REGION Network 4: Alarm_GlobalError SubStation and RemoteIO
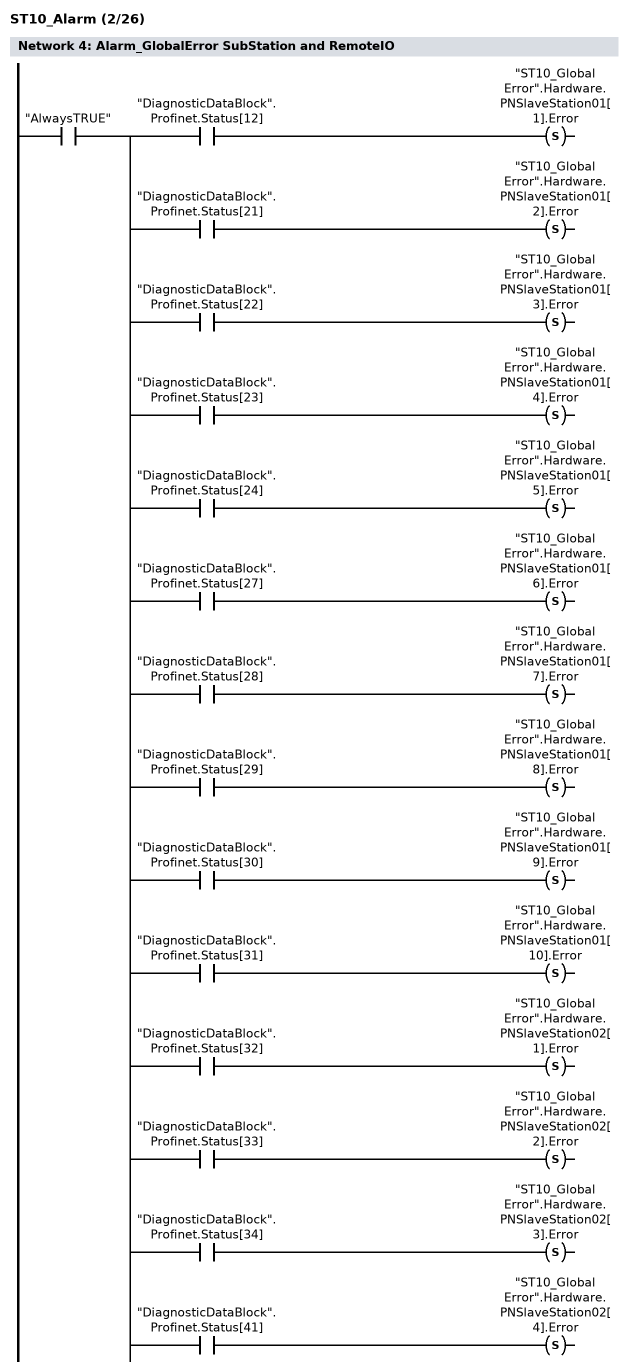
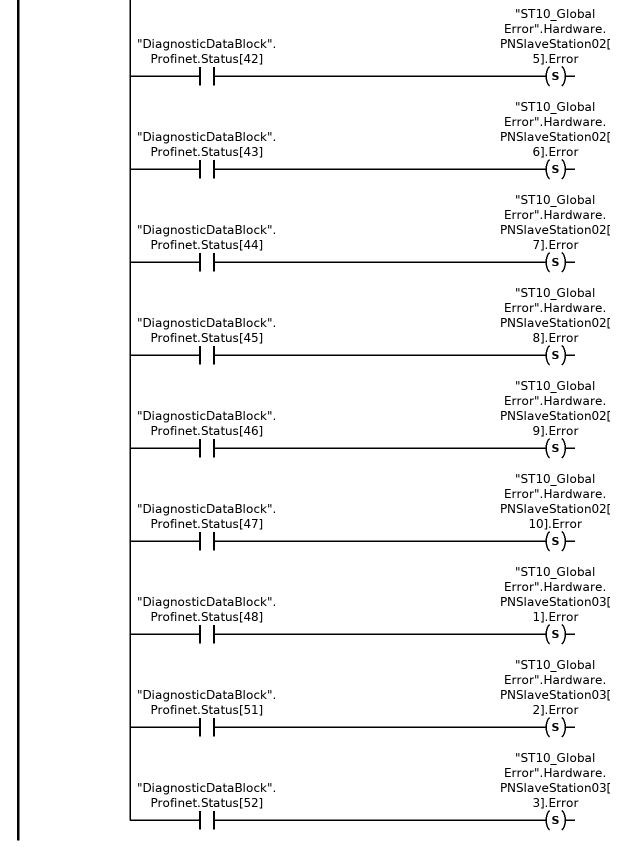
   RUNG wire#powerrail
      Contact( "AlwaysTRUE" )
      wire#w1
      Contact( "DiagnosticDataBlock".Profinet.Status[12] )
      S_Coil( "ST10_GlobalError".Hardware.PNSlaveStation01[1].Error )
   END_RUNG
   RUNG wire#w1
      Contact( "DiagnosticDataBlock".Profinet.Status[21] )
      S_Coil( "ST10_GlobalError".Hardware.PNSlaveStation01[2].Error )
   END_RUNG
   RUNG wire#w1
      Contact( "DiagnosticDataBlock".Profinet.Status[22] )
      S_Coil( "ST10_GlobalError".Hardware.PNSlaveStation01[3].Error )
   END_RUNG
   RUNG wire#w1
      Contact( "DiagnosticDataBlock".Profinet.Status[23] )
      S_Coil( "ST10_GlobalError".Hardware.PNSlaveStation01[4].Error )
   END_RUNG
   RUNG wire#w1
      Contact( "DiagnosticDataBlock".Profinet.Status[24] )
      S_Coil( "ST10_GlobalError".Hardware.PNSlaveStation01[5].Error )
   END_RUNG
   RUNG wire#w1
      Contact( "DiagnosticDataBlock".Profinet.Status[27] )
      S_Coil( "ST10_GlobalError".Hardware.PNSlaveStation01[6].Error )
   END_RUNG
   RUNG wire#w1
      Contact( "DiagnosticDataBlock".Profinet.Status[28] )
      S_Coil( "ST10_GlobalError".Hardware.PNSlaveStation01[7].Error )
   END_RUNG
   RUNG wire#w1
      Contact( "DiagnosticDataBlock".Profinet.Status[29] )
      S_Coil( "ST10_GlobalError".Hardware.PNSlaveStation01[8].Error )
   END_RUNG
   RUNG wire#w1
      Contact( "DiagnosticDataBlock".Profinet.Status[30] )
      S_Coil( "ST10_GlobalError".Hardware.PNSlaveStation01[9].Error )
   END_RUNG
   RUNG wire#w1
      Contact( "DiagnosticDataBlock".Profinet.Status[31] )
      S_Coil( "ST10_GlobalError".Hardware.PNSlaveStation01[10].Error )
   END_RUNG
   RUNG wire#w1
      Contact( "DiagnosticDataBlock".Profinet.Status[32] )
      S_Coil( "ST10_GlobalError".Hardware.PNSlaveStation02[1].Error )
   END_RUNG
   RUNG wire#w1
      Contact( "DiagnosticDataBlock".Profinet.Status[33] )
      S_Coil( "ST10_GlobalError".Hardware.PNSlaveStation02[2].Error )
   END_RUNG
   RUNG wire#w1
      Contact( "DiagnosticDataBlock".Profinet.Status[34] )
      S_Coil( "ST10_GlobalError".Hardware.PNSlaveStation02[3].Error )
   END_RUNG
   RUNG wire#w1
      Contact( "DiagnosticDataBlock".Profinet.Status[41] )
      S_Coil( "ST10_GlobalError".Hardware.PNSlaveStation02[4].Error )
   END_RUNG
   RUNG wire#w1
      Contact( "DiagnosticDataBlock".Profinet.Status[42] )
      S_Coil( "ST10_GlobalError".Hardware.PNSlaveStation02[5].Error )
   END_RUNG
   RUNG wire#w1
      Contact( "DiagnosticDataBlock".Profinet.Status[43] )
      S_Coil( "ST10_GlobalError".Hardware.PNSlaveStation02[6].Error )
   END_RUNG
   RUNG wire#w1
      Contact( "DiagnosticDataBlock".Profinet.Status[44] )
      S_Coil( "ST10_GlobalError".Hardware.PNSlaveStation02[7].Error )
   END_RUNG
   RUNG wire#w1
      Contact( "DiagnosticDataBlock".Profinet.Status[45] )
      S_Coil( "ST10_GlobalError".Hardware.PNSlaveStation02[8].Error )
   END_RUNG
   RUNG wire#w1
      Contact( "DiagnosticDataBlock".Profinet.Status[46] )
      S_Coil( "ST10_GlobalError".Hardware.PNSlaveStation02[9].Error )
   END_RUNG
   RUNG wire#w1
      Contact( "DiagnosticDataBlock".Profinet.Status[47] )
      S_Coil( "ST10_GlobalError".Hardware.PNSlaveStation02[10].Error )
   END_RUNG
   RUNG wire#w1
      Contact( "DiagnosticDataBlock".Profinet.Status[48] )
      S_Coil( "ST10_GlobalError".Hardware.PNSlaveStation03[1].Error )
   END_RUNG
   RUNG wire#w1
      Contact( "DiagnosticDataBlock".Profinet.Status[51] )
      S_Coil( "ST10_GlobalError".Hardware.PNSlaveStation03[2].Error )
   END_RUNG
   RUNG wire#w1
      Contact( "DiagnosticDataBlock".Profinet.Status[52] )
      S_Coil( "ST10_GlobalError".Hardware.PNSlaveStation03[3].Error )
   END_RUNG
   // the same network as SCL:
   IF "AlwaysTRUE" AND "DiagnosticDataBlock".Profinet.Status[12] THEN
       "ST10_GlobalError".Hardware.PNSlaveStation01[1].Error := TRUE;
   END_IF;
   IF "AlwaysTRUE" AND "DiagnosticDataBlock".Profinet.Status[21] THEN
       "ST10_GlobalError".Hardware.PNSlaveStation01[2].Error := TRUE;
   END_IF;
   IF "AlwaysTRUE" AND "DiagnosticDataBlock".Profinet.Status[22] THEN
       "ST10_GlobalError".Hardware.PNSlaveStation01[3].Error := TRUE;
   END_IF;
   IF "AlwaysTRUE" AND "DiagnosticDataBlock".Profinet.Status[23] THEN
       "ST10_GlobalError".Hardware.PNSlaveStation01[4].Error := TRUE;
   END_IF;
   IF "AlwaysTRUE" AND "DiagnosticDataBlock".Profinet.Status[24] THEN
       "ST10_GlobalError".Hardware.PNSlaveStation01[5].Error := TRUE;
   END_IF;
   IF "AlwaysTRUE" AND "DiagnosticDataBlock".Profinet.Status[27] THEN
       "ST10_GlobalError".Hardware.PNSlaveStation01[6].Error := TRUE;
   END_IF;
   IF "AlwaysTRUE" AND "DiagnosticDataBlock".Profinet.Status[28] THEN
       "ST10_GlobalError".Hardware.PNSlaveStation01[7].Error := TRUE;
   END_IF;
   IF "AlwaysTRUE" AND "DiagnosticDataBlock".Profinet.Status[29] THEN
       "ST10_GlobalError".Hardware.PNSlaveStation01[8].Error := TRUE;
   END_IF;
   IF "AlwaysTRUE" AND "DiagnosticDataBlock".Profinet.Status[30] THEN
       "ST10_GlobalError".Hardware.PNSlaveStation01[9].Error := TRUE;
   END_IF;
   IF "AlwaysTRUE" AND "DiagnosticDataBlock".Profinet.Status[31] THEN
       "ST10_GlobalError".Hardware.PNSlaveStation01[10].Error := TRUE;
   END_IF;
   IF "AlwaysTRUE" AND "DiagnosticDataBlock".Profinet.Status[32] THEN
       "ST10_GlobalError".Hardware.PNSlaveStation02[1].Error := TRUE;
   END_IF;
   IF "AlwaysTRUE" AND "DiagnosticDataBlock".Profinet.Status[33] THEN
       "ST10_GlobalError".Hardware.PNSlaveStation02[2].Error := TRUE;
   END_IF;
   IF "AlwaysTRUE" AND "DiagnosticDataBlock".Profinet.Status[34] THEN
       "ST10_GlobalError".Hardware.PNSlaveStation02[3].Error := TRUE;
   END_IF;
   IF "AlwaysTRUE" AND "DiagnosticDataBlock".Profinet.Status[41] THEN
       "ST10_GlobalError".Hardware.PNSlaveStation02[4].Error := TRUE;
   END_IF;
   IF "AlwaysTRUE" AND "DiagnosticDataBlock".Profinet.Status[42] THEN
       "ST10_GlobalError".Hardware.PNSlaveStation02[5].Error := TRUE;
   END_IF;
   IF "AlwaysTRUE" AND "DiagnosticDataBlock".Profinet.Status[43] THEN
       "ST10_GlobalError".Hardware.PNSlaveStation02[6].Error := TRUE;
   END_IF;
   IF "AlwaysTRUE" AND "DiagnosticDataBlock".Profinet.Status[44] THEN
       "ST10_GlobalError".Hardware.PNSlaveStation02[7].Error := TRUE;
   END_IF;
   IF "AlwaysTRUE" AND "DiagnosticDataBlock".Profinet.Status[45] THEN
       "ST10_GlobalError".Hardware.PNSlaveStation02[8].Error := TRUE;
   END_IF;
   IF "AlwaysTRUE" AND "DiagnosticDataBlock".Profinet.Status[46] THEN
       "ST10_GlobalError".Hardware.PNSlaveStation02[9].Error := TRUE;
   END_IF;
   IF "AlwaysTRUE" AND "DiagnosticDataBlock".Profinet.Status[47] THEN
       "ST10_GlobalError".Hardware.PNSlaveStation02[10].Error := TRUE;
   END_IF;
   IF "AlwaysTRUE" AND "DiagnosticDataBlock".Profinet.Status[48] THEN
       "ST10_GlobalError".Hardware.PNSlaveStation03[1].Error := TRUE;
   END_IF;
   IF "AlwaysTRUE" AND "DiagnosticDataBlock".Profinet.Status[51] THEN
       "ST10_GlobalError".Hardware.PNSlaveStation03[2].Error := TRUE;
   END_IF;
   IF "AlwaysTRUE" AND "DiagnosticDataBlock".Profinet.Status[52] THEN
       "ST10_GlobalError".Hardware.PNSlaveStation03[3].Error := TRUE;
   END_IF;
END_REGION

REGION Network 5: Alarm_GlobalError Valve island
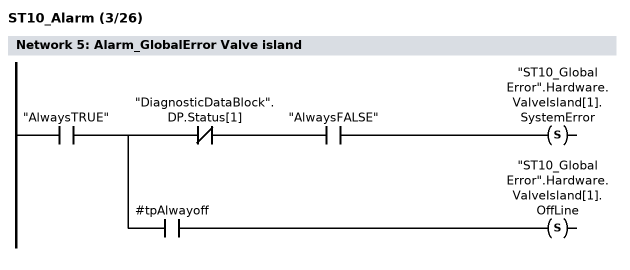
   RUNG wire#powerrail
      Contact( "AlwaysTRUE" )
      wire#w1
      I_Contact( "DiagnosticDataBlock".DP.Status[1] )
      Contact( "AlwaysFALSE" )
      S_Coil( "ST10_GlobalError".Hardware.ValveIsland[1].SystemError )
   END_RUNG
   RUNG wire#w1
      Contact( #tpAlwayoff )
      S_Coil( "ST10_GlobalError".Hardware.ValveIsland[1].OffLine )
   END_RUNG
   // the same network as SCL:
   IF "AlwaysTRUE" AND NOT "DiagnosticDataBlock".DP.Status[1] AND "AlwaysFALSE" THEN
       "ST10_GlobalError".Hardware.ValveIsland[1].SystemError := TRUE;
   END_IF;
   IF "AlwaysTRUE" AND #tpAlwayoff THEN "ST10_GlobalError".Hardware.ValveIsland[1].OffLine := TRUE; END_IF;
END_REGION

REGION Network 6: Alarm_GlobalError Safety Circuit and E-stop
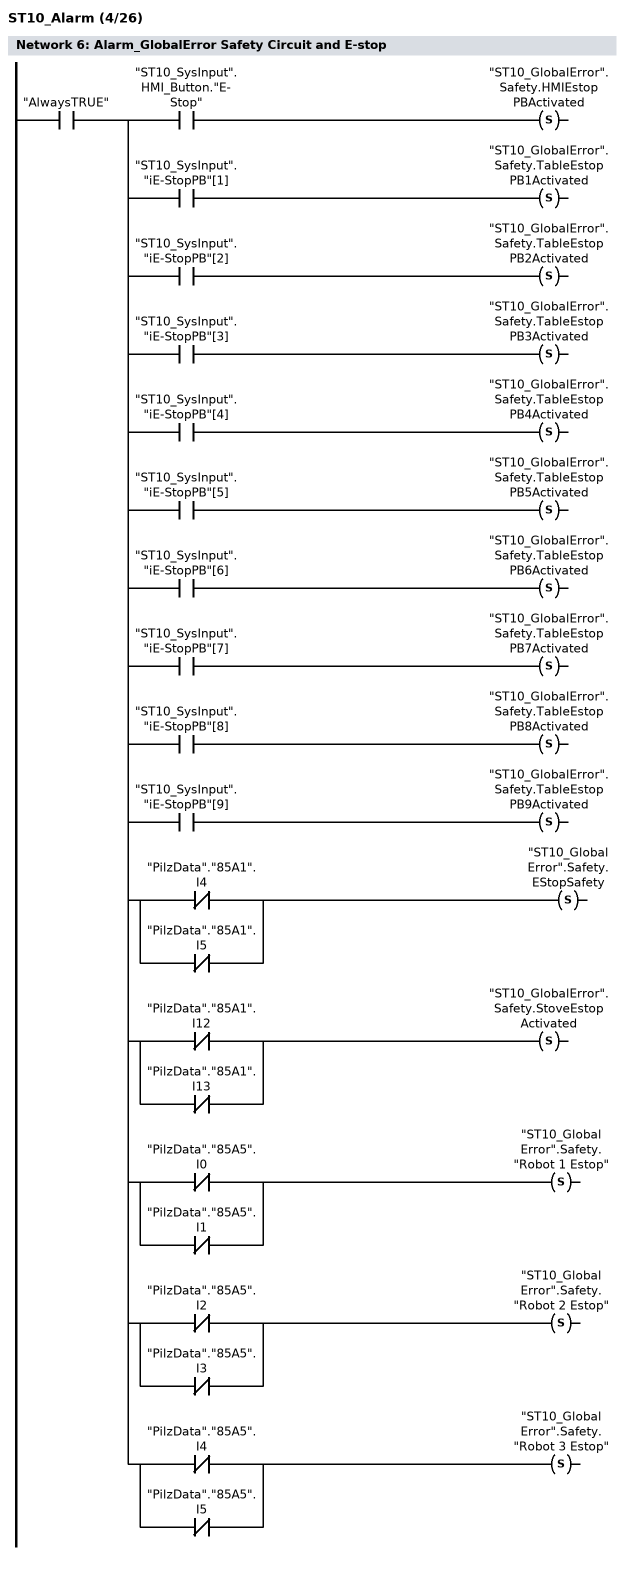
   RUNG wire#powerrail
      Contact( "AlwaysTRUE" )
      wire#w1
      Contact( "ST10_SysInput".HMI_Button."E-Stop" )
      S_Coil( "ST10_GlobalError".Safety.HMIEstopPBActivated )
   END_RUNG
   RUNG wire#w1
      Contact( "ST10_SysInput"."iE-StopPB"[1] )
      S_Coil( "ST10_GlobalError".Safety.TableEstopPB1Activated )
   END_RUNG
   RUNG wire#w1
      Contact( "ST10_SysInput"."iE-StopPB"[2] )
      S_Coil( "ST10_GlobalError".Safety.TableEstopPB2Activated )
   END_RUNG
   RUNG wire#w1
      Contact( "ST10_SysInput"."iE-StopPB"[3] )
      S_Coil( "ST10_GlobalError".Safety.TableEstopPB3Activated )
   END_RUNG
   RUNG wire#w1
      Contact( "ST10_SysInput"."iE-StopPB"[4] )
      S_Coil( "ST10_GlobalError".Safety.TableEstopPB4Activated )
   END_RUNG
   RUNG wire#w1
      Contact( "ST10_SysInput"."iE-StopPB"[5] )
      S_Coil( "ST10_GlobalError".Safety.TableEstopPB5Activated )
   END_RUNG
   RUNG wire#w1
      Contact( "ST10_SysInput"."iE-StopPB"[6] )
      S_Coil( "ST10_GlobalError".Safety.TableEstopPB6Activated )
   END_RUNG
   RUNG wire#w1
      Contact( "ST10_SysInput"."iE-StopPB"[7] )
      S_Coil( "ST10_GlobalError".Safety.TableEstopPB7Activated )
   END_RUNG
   RUNG wire#w1
      Contact( "ST10_SysInput"."iE-StopPB"[8] )
      S_Coil( "ST10_GlobalError".Safety.TableEstopPB8Activated )
   END_RUNG
   RUNG wire#w1
      Contact( "ST10_SysInput"."iE-StopPB"[9] )
      S_Coil( "ST10_GlobalError".Safety.TableEstopPB9Activated )
   END_RUNG
   RUNG wire#w1
      I_Contact( "PilzData"."85A1".I4 )
      wire#w2
      S_Coil( "ST10_GlobalError".Safety.EStopSafety )
   END_RUNG
   RUNG wire#w1
      I_Contact( "PilzData"."85A1".I5 )
   END_RUNG wire#w2
   RUNG wire#w1
      I_Contact( "PilzData"."85A1".I12 )
      wire#w3
      S_Coil( "ST10_GlobalError".Safety.StoveEstopActivated )
   END_RUNG
   RUNG wire#w1
      I_Contact( "PilzData"."85A1".I13 )
   END_RUNG wire#w3
   RUNG wire#w1
      I_Contact( "PilzData"."85A5".I0 )
      wire#w4
      S_Coil( "ST10_GlobalError".Safety."Robot 1 Estop" )
   END_RUNG
   RUNG wire#w1
      I_Contact( "PilzData"."85A5".I1 )
   END_RUNG wire#w4
   RUNG wire#w1
      I_Contact( "PilzData"."85A5".I2 )
      wire#w5
      S_Coil( "ST10_GlobalError".Safety."Robot 2 Estop" )
   END_RUNG
   RUNG wire#w1
      I_Contact( "PilzData"."85A5".I3 )
   END_RUNG wire#w5
   RUNG wire#w1
      I_Contact( "PilzData"."85A5".I4 )
      wire#w6
      S_Coil( "ST10_GlobalError".Safety."Robot 3 Estop" )
   END_RUNG
   RUNG wire#w1
      I_Contact( "PilzData"."85A5".I5 )
   END_RUNG wire#w6
   // the same network as SCL:
   IF "AlwaysTRUE" AND "ST10_SysInput".HMI_Button."E-Stop" THEN
       "ST10_GlobalError".Safety.HMIEstopPBActivated := TRUE;
   END_IF;
   IF "AlwaysTRUE" AND "ST10_SysInput"."iE-StopPB"[1] THEN
       "ST10_GlobalError".Safety.TableEstopPB1Activated := TRUE;
   END_IF;
   IF "AlwaysTRUE" AND "ST10_SysInput"."iE-StopPB"[2] THEN
       "ST10_GlobalError".Safety.TableEstopPB2Activated := TRUE;
   END_IF;
   IF "AlwaysTRUE" AND "ST10_SysInput"."iE-StopPB"[3] THEN
       "ST10_GlobalError".Safety.TableEstopPB3Activated := TRUE;
   END_IF;
   IF "AlwaysTRUE" AND "ST10_SysInput"."iE-StopPB"[4] THEN
       "ST10_GlobalError".Safety.TableEstopPB4Activated := TRUE;
   END_IF;
   IF "AlwaysTRUE" AND "ST10_SysInput"."iE-StopPB"[5] THEN
       "ST10_GlobalError".Safety.TableEstopPB5Activated := TRUE;
   END_IF;
   IF "AlwaysTRUE" AND "ST10_SysInput"."iE-StopPB"[6] THEN
       "ST10_GlobalError".Safety.TableEstopPB6Activated := TRUE;
   END_IF;
   IF "AlwaysTRUE" AND "ST10_SysInput"."iE-StopPB"[7] THEN
       "ST10_GlobalError".Safety.TableEstopPB7Activated := TRUE;
   END_IF;
   IF "AlwaysTRUE" AND "ST10_SysInput"."iE-StopPB"[8] THEN
       "ST10_GlobalError".Safety.TableEstopPB8Activated := TRUE;
   END_IF;
   IF "AlwaysTRUE" AND "ST10_SysInput"."iE-StopPB"[9] THEN
       "ST10_GlobalError".Safety.TableEstopPB9Activated := TRUE;
   END_IF;
   IF "AlwaysTRUE" AND (NOT "PilzData"."85A1".I4 OR NOT "PilzData"."85A1".I5) THEN
       "ST10_GlobalError".Safety.EStopSafety := TRUE;
   END_IF;
   IF "AlwaysTRUE" AND (NOT "PilzData"."85A1".I12 OR NOT "PilzData"."85A1".I13) THEN
       "ST10_GlobalError".Safety.StoveEstopActivated := TRUE;
   END_IF;
   IF "AlwaysTRUE" AND (NOT "PilzData"."85A5".I0 OR NOT "PilzData"."85A5".I1) THEN
       "ST10_GlobalError".Safety."Robot 1 Estop" := TRUE;
   END_IF;
   IF "AlwaysTRUE" AND (NOT "PilzData"."85A5".I2 OR NOT "PilzData"."85A5".I3) THEN
       "ST10_GlobalError".Safety."Robot 2 Estop" := TRUE;
   END_IF;
   IF "AlwaysTRUE" AND (NOT "PilzData"."85A5".I4 OR NOT "PilzData"."85A5".I5) THEN
       "ST10_GlobalError".Safety."Robot 3 Estop" := TRUE;
   END_IF;
END_REGION

REGION Network 7: Alarm_GlobalError Safety Door / Alarm_GlobalError Safety Door 110-124
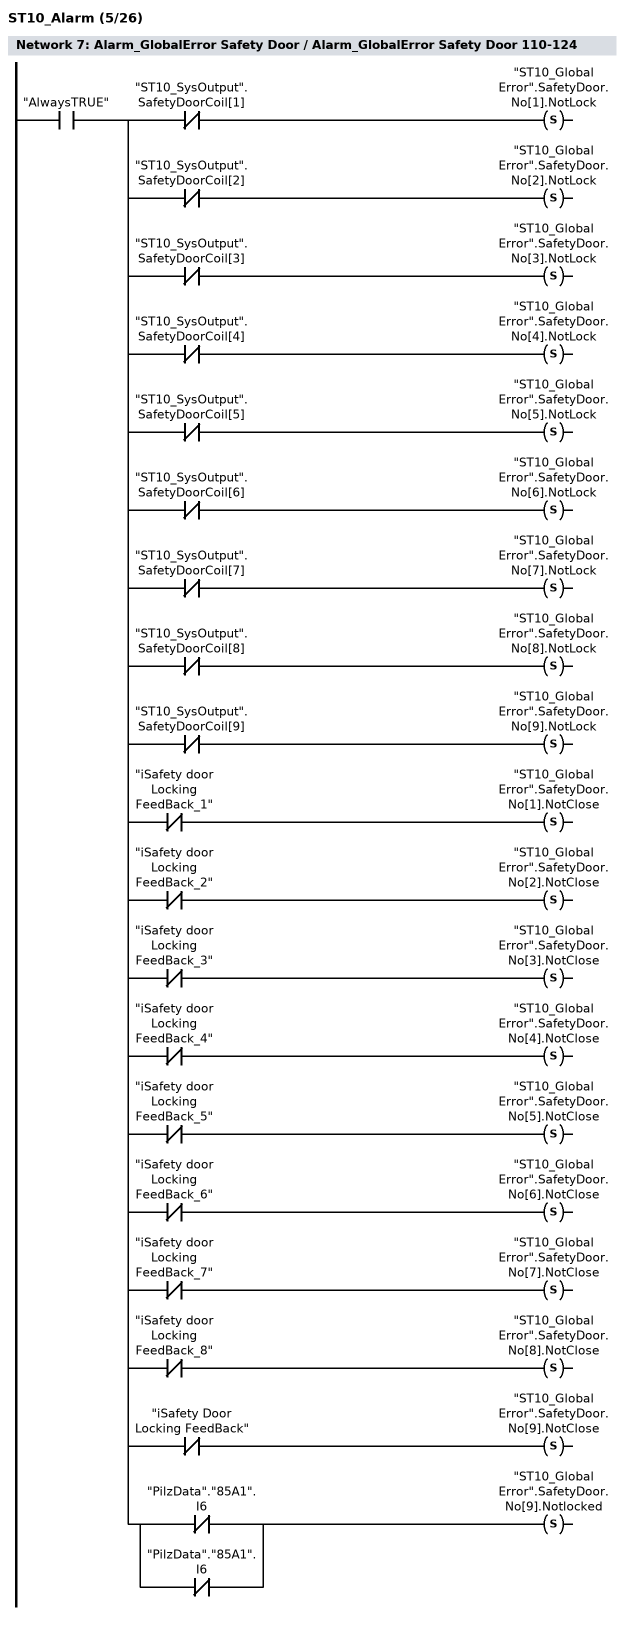
   RUNG wire#powerrail
      Contact( "AlwaysTRUE" )
      wire#w1
      I_Contact( "ST10_SysOutput".SafetyDoorCoil[1] )
      S_Coil( "ST10_GlobalError".SafetyDoor.No[1].NotLock )
   END_RUNG
   RUNG wire#w1
      I_Contact( "ST10_SysOutput".SafetyDoorCoil[2] )
      S_Coil( "ST10_GlobalError".SafetyDoor.No[2].NotLock )
   END_RUNG
   RUNG wire#w1
      I_Contact( "ST10_SysOutput".SafetyDoorCoil[3] )
      S_Coil( "ST10_GlobalError".SafetyDoor.No[3].NotLock )
   END_RUNG
   RUNG wire#w1
      I_Contact( "ST10_SysOutput".SafetyDoorCoil[4] )
      S_Coil( "ST10_GlobalError".SafetyDoor.No[4].NotLock )
   END_RUNG
   RUNG wire#w1
      I_Contact( "ST10_SysOutput".SafetyDoorCoil[5] )
      S_Coil( "ST10_GlobalError".SafetyDoor.No[5].NotLock )
   END_RUNG
   RUNG wire#w1
      I_Contact( "ST10_SysOutput".SafetyDoorCoil[6] )
      S_Coil( "ST10_GlobalError".SafetyDoor.No[6].NotLock )
   END_RUNG
   RUNG wire#w1
      I_Contact( "ST10_SysOutput".SafetyDoorCoil[7] )
      S_Coil( "ST10_GlobalError".SafetyDoor.No[7].NotLock )
   END_RUNG
   RUNG wire#w1
      I_Contact( "ST10_SysOutput".SafetyDoorCoil[8] )
      S_Coil( "ST10_GlobalError".SafetyDoor.No[8].NotLock )
   END_RUNG
   RUNG wire#w1
      I_Contact( "ST10_SysOutput".SafetyDoorCoil[9] )
      S_Coil( "ST10_GlobalError".SafetyDoor.No[9].NotLock )
   END_RUNG
   RUNG wire#w1
      I_Contact( "iSafety door Locking FeedBack_1" )
      S_Coil( "ST10_GlobalError".SafetyDoor.No[1].NotClose )
   END_RUNG
   RUNG wire#w1
      I_Contact( "iSafety door Locking FeedBack_2" )
      S_Coil( "ST10_GlobalError".SafetyDoor.No[2].NotClose )
   END_RUNG
   RUNG wire#w1
      I_Contact( "iSafety door Locking FeedBack_3" )
      S_Coil( "ST10_GlobalError".SafetyDoor.No[3].NotClose )
   END_RUNG
   RUNG wire#w1
      I_Contact( "iSafety door Locking FeedBack_4" )
      S_Coil( "ST10_GlobalError".SafetyDoor.No[4].NotClose )
   END_RUNG
   RUNG wire#w1
      I_Contact( "iSafety door Locking FeedBack_5" )
      S_Coil( "ST10_GlobalError".SafetyDoor.No[5].NotClose )
   END_RUNG
   RUNG wire#w1
      I_Contact( "iSafety door Locking FeedBack_6" )
      S_Coil( "ST10_GlobalError".SafetyDoor.No[6].NotClose )
   END_RUNG
   RUNG wire#w1
      I_Contact( "iSafety door Locking FeedBack_7" )
      S_Coil( "ST10_GlobalError".SafetyDoor.No[7].NotClose )
   END_RUNG
   RUNG wire#w1
      I_Contact( "iSafety door Locking FeedBack_8" )
      S_Coil( "ST10_GlobalError".SafetyDoor.No[8].NotClose )
   END_RUNG
   RUNG wire#w1
      I_Contact( "iSafety Door Locking FeedBack" )
      S_Coil( "ST10_GlobalError".SafetyDoor.No[9].NotClose )
   END_RUNG
   RUNG wire#w1
      I_Contact( "PilzData"."85A1".I6 )
      wire#w2
      S_Coil( "ST10_GlobalError".SafetyDoor.No[9].Notlocked )
   END_RUNG
   RUNG wire#w1
      I_Contact( "PilzData"."85A1".I6 )
   END_RUNG wire#w2
   // the same network as SCL:
   IF "AlwaysTRUE" AND NOT "ST10_SysOutput".SafetyDoorCoil[1] THEN
       "ST10_GlobalError".SafetyDoor.No[1].NotLock := TRUE;
   END_IF;
   IF "AlwaysTRUE" AND NOT "ST10_SysOutput".SafetyDoorCoil[2] THEN
       "ST10_GlobalError".SafetyDoor.No[2].NotLock := TRUE;
   END_IF;
   IF "AlwaysTRUE" AND NOT "ST10_SysOutput".SafetyDoorCoil[3] THEN
       "ST10_GlobalError".SafetyDoor.No[3].NotLock := TRUE;
   END_IF;
   IF "AlwaysTRUE" AND NOT "ST10_SysOutput".SafetyDoorCoil[4] THEN
       "ST10_GlobalError".SafetyDoor.No[4].NotLock := TRUE;
   END_IF;
   IF "AlwaysTRUE" AND NOT "ST10_SysOutput".SafetyDoorCoil[5] THEN
       "ST10_GlobalError".SafetyDoor.No[5].NotLock := TRUE;
   END_IF;
   IF "AlwaysTRUE" AND NOT "ST10_SysOutput".SafetyDoorCoil[6] THEN
       "ST10_GlobalError".SafetyDoor.No[6].NotLock := TRUE;
   END_IF;
   IF "AlwaysTRUE" AND NOT "ST10_SysOutput".SafetyDoorCoil[7] THEN
       "ST10_GlobalError".SafetyDoor.No[7].NotLock := TRUE;
   END_IF;
   IF "AlwaysTRUE" AND NOT "ST10_SysOutput".SafetyDoorCoil[8] THEN
       "ST10_GlobalError".SafetyDoor.No[8].NotLock := TRUE;
   END_IF;
   IF "AlwaysTRUE" AND NOT "ST10_SysOutput".SafetyDoorCoil[9] THEN
       "ST10_GlobalError".SafetyDoor.No[9].NotLock := TRUE;
   END_IF;
   IF "AlwaysTRUE" AND NOT "iSafety door Locking FeedBack_1" THEN
       "ST10_GlobalError".SafetyDoor.No[1].NotClose := TRUE;
   END_IF;
   IF "AlwaysTRUE" AND NOT "iSafety door Locking FeedBack_2" THEN
       "ST10_GlobalError".SafetyDoor.No[2].NotClose := TRUE;
   END_IF;
   IF "AlwaysTRUE" AND NOT "iSafety door Locking FeedBack_3" THEN
       "ST10_GlobalError".SafetyDoor.No[3].NotClose := TRUE;
   END_IF;
   IF "AlwaysTRUE" AND NOT "iSafety door Locking FeedBack_4" THEN
       "ST10_GlobalError".SafetyDoor.No[4].NotClose := TRUE;
   END_IF;
   IF "AlwaysTRUE" AND NOT "iSafety door Locking FeedBack_5" THEN
       "ST10_GlobalError".SafetyDoor.No[5].NotClose := TRUE;
   END_IF;
   IF "AlwaysTRUE" AND NOT "iSafety door Locking FeedBack_6" THEN
       "ST10_GlobalError".SafetyDoor.No[6].NotClose := TRUE;
   END_IF;
   IF "AlwaysTRUE" AND NOT "iSafety door Locking FeedBack_7" THEN
       "ST10_GlobalError".SafetyDoor.No[7].NotClose := TRUE;
   END_IF;
   IF "AlwaysTRUE" AND NOT "iSafety door Locking FeedBack_8" THEN
       "ST10_GlobalError".SafetyDoor.No[8].NotClose := TRUE;
   END_IF;
   IF "AlwaysTRUE" AND NOT "iSafety Door Locking FeedBack" THEN
       "ST10_GlobalError".SafetyDoor.No[9].NotClose := TRUE;
   END_IF;
   IF "AlwaysTRUE" AND (NOT "PilzData"."85A1".I6 OR NOT "PilzData"."85A1".I6) THEN
       "ST10_GlobalError".SafetyDoor.No[9].Notlocked := TRUE;
   END_IF;
END_REGION

REGION Network 8: Alarm_GlobalError Safety Door / Alarm_GlobalError Material Door 128-129
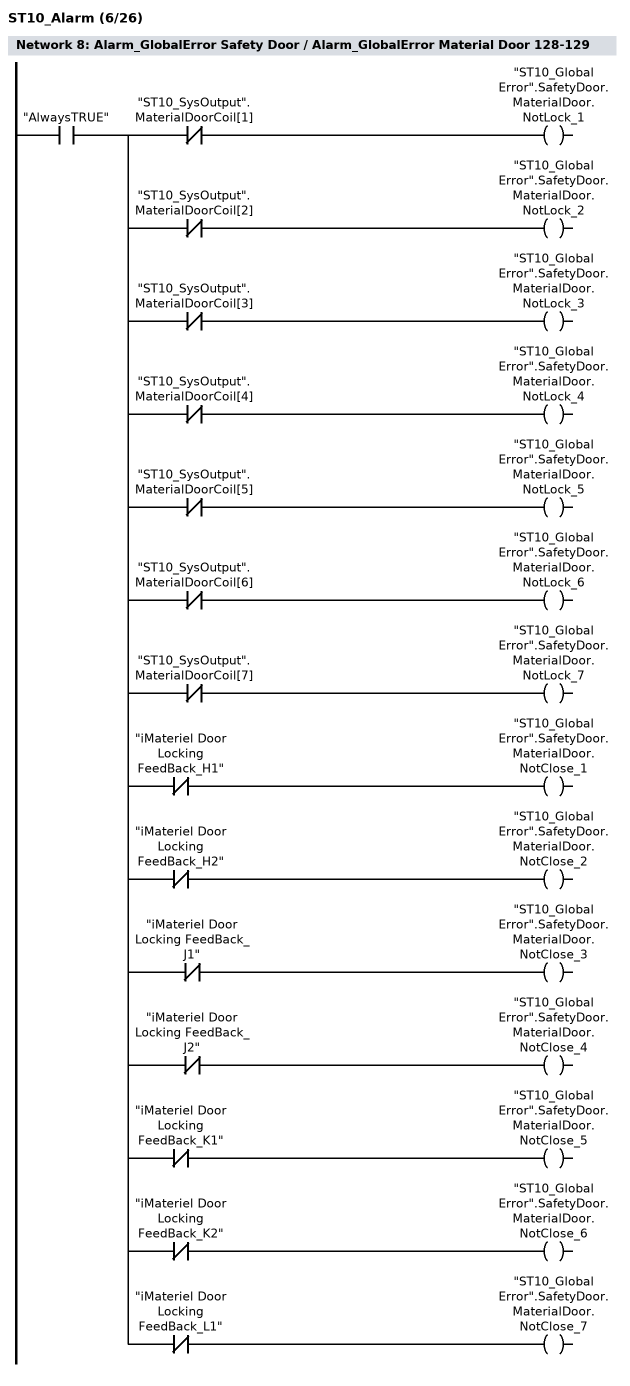
   RUNG wire#powerrail
      Contact( "AlwaysTRUE" )
      wire#w1
      I_Contact( "ST10_SysOutput".MaterialDoorCoil[1] )
      Coil( "ST10_GlobalError".SafetyDoor.MaterialDoor.NotLock_1 )
   END_RUNG
   RUNG wire#w1
      I_Contact( "ST10_SysOutput".MaterialDoorCoil[2] )
      Coil( "ST10_GlobalError".SafetyDoor.MaterialDoor.NotLock_2 )
   END_RUNG
   RUNG wire#w1
      I_Contact( "ST10_SysOutput".MaterialDoorCoil[3] )
      Coil( "ST10_GlobalError".SafetyDoor.MaterialDoor.NotLock_3 )
   END_RUNG
   RUNG wire#w1
      I_Contact( "ST10_SysOutput".MaterialDoorCoil[4] )
      Coil( "ST10_GlobalError".SafetyDoor.MaterialDoor.NotLock_4 )
   END_RUNG
   RUNG wire#w1
      I_Contact( "ST10_SysOutput".MaterialDoorCoil[5] )
      Coil( "ST10_GlobalError".SafetyDoor.MaterialDoor.NotLock_5 )
   END_RUNG
   RUNG wire#w1
      I_Contact( "ST10_SysOutput".MaterialDoorCoil[6] )
      Coil( "ST10_GlobalError".SafetyDoor.MaterialDoor.NotLock_6 )
   END_RUNG
   RUNG wire#w1
      I_Contact( "ST10_SysOutput".MaterialDoorCoil[7] )
      Coil( "ST10_GlobalError".SafetyDoor.MaterialDoor.NotLock_7 )
   END_RUNG
   RUNG wire#w1
      I_Contact( "iMateriel Door Locking FeedBack_H1" )
      Coil( "ST10_GlobalError".SafetyDoor.MaterialDoor.NotClose_1 )
   END_RUNG
   RUNG wire#w1
      I_Contact( "iMateriel Door Locking FeedBack_H2" )
      Coil( "ST10_GlobalError".SafetyDoor.MaterialDoor.NotClose_2 )
   END_RUNG
   RUNG wire#w1
      I_Contact( "iMateriel Door Locking FeedBack_J1" )
      Coil( "ST10_GlobalError".SafetyDoor.MaterialDoor.NotClose_3 )
   END_RUNG
   RUNG wire#w1
      I_Contact( "iMateriel Door Locking FeedBack_J2" )
      Coil( "ST10_GlobalError".SafetyDoor.MaterialDoor.NotClose_4 )
   END_RUNG
   RUNG wire#w1
      I_Contact( "iMateriel Door Locking FeedBack_K1" )
      Coil( "ST10_GlobalError".SafetyDoor.MaterialDoor.NotClose_5 )
   END_RUNG
   RUNG wire#w1
      I_Contact( "iMateriel Door Locking FeedBack_K2" )
      Coil( "ST10_GlobalError".SafetyDoor.MaterialDoor.NotClose_6 )
   END_RUNG
   RUNG wire#w1
      I_Contact( "iMateriel Door Locking FeedBack_L1" )
      Coil( "ST10_GlobalError".SafetyDoor.MaterialDoor.NotClose_7 )
   END_RUNG
   // the same network as SCL:
   "ST10_GlobalError".SafetyDoor.MaterialDoor.NotLock_1 := "AlwaysTRUE" AND NOT "ST10_SysOutput".MaterialDoorCoil[1];
   "ST10_GlobalError".SafetyDoor.MaterialDoor.NotLock_2 := "AlwaysTRUE" AND NOT "ST10_SysOutput".MaterialDoorCoil[2];
   "ST10_GlobalError".SafetyDoor.MaterialDoor.NotLock_3 := "AlwaysTRUE" AND NOT "ST10_SysOutput".MaterialDoorCoil[3];
   "ST10_GlobalError".SafetyDoor.MaterialDoor.NotLock_4 := "AlwaysTRUE" AND NOT "ST10_SysOutput".MaterialDoorCoil[4];
   "ST10_GlobalError".SafetyDoor.MaterialDoor.NotLock_5 := "AlwaysTRUE" AND NOT "ST10_SysOutput".MaterialDoorCoil[5];
   "ST10_GlobalError".SafetyDoor.MaterialDoor.NotLock_6 := "AlwaysTRUE" AND NOT "ST10_SysOutput".MaterialDoorCoil[6];
   "ST10_GlobalError".SafetyDoor.MaterialDoor.NotLock_7 := "AlwaysTRUE" AND NOT "ST10_SysOutput".MaterialDoorCoil[7];
   "ST10_GlobalError".SafetyDoor.MaterialDoor.NotClose_1 := "AlwaysTRUE" AND NOT "iMateriel Door Locking FeedBack_H1";
   "ST10_GlobalError".SafetyDoor.MaterialDoor.NotClose_2 := "AlwaysTRUE" AND NOT "iMateriel Door Locking FeedBack_H2";
   "ST10_GlobalError".SafetyDoor.MaterialDoor.NotClose_3 := "AlwaysTRUE" AND NOT "iMateriel Door Locking FeedBack_J1";
   "ST10_GlobalError".SafetyDoor.MaterialDoor.NotClose_4 := "AlwaysTRUE" AND NOT "iMateriel Door Locking FeedBack_J2";
   "ST10_GlobalError".SafetyDoor.MaterialDoor.NotClose_5 := "AlwaysTRUE" AND NOT "iMateriel Door Locking FeedBack_K1";
   "ST10_GlobalError".SafetyDoor.MaterialDoor.NotClose_6 := "AlwaysTRUE" AND NOT "iMateriel Door Locking FeedBack_K2";
   "ST10_GlobalError".SafetyDoor.MaterialDoor.NotClose_7 := "AlwaysTRUE" AND NOT "iMateriel Door Locking FeedBack_L1";
END_REGION

REGION Network 9: Alarm_GlobalError Safety Door / Alarm_GlobalError Material Door Safety 128-129
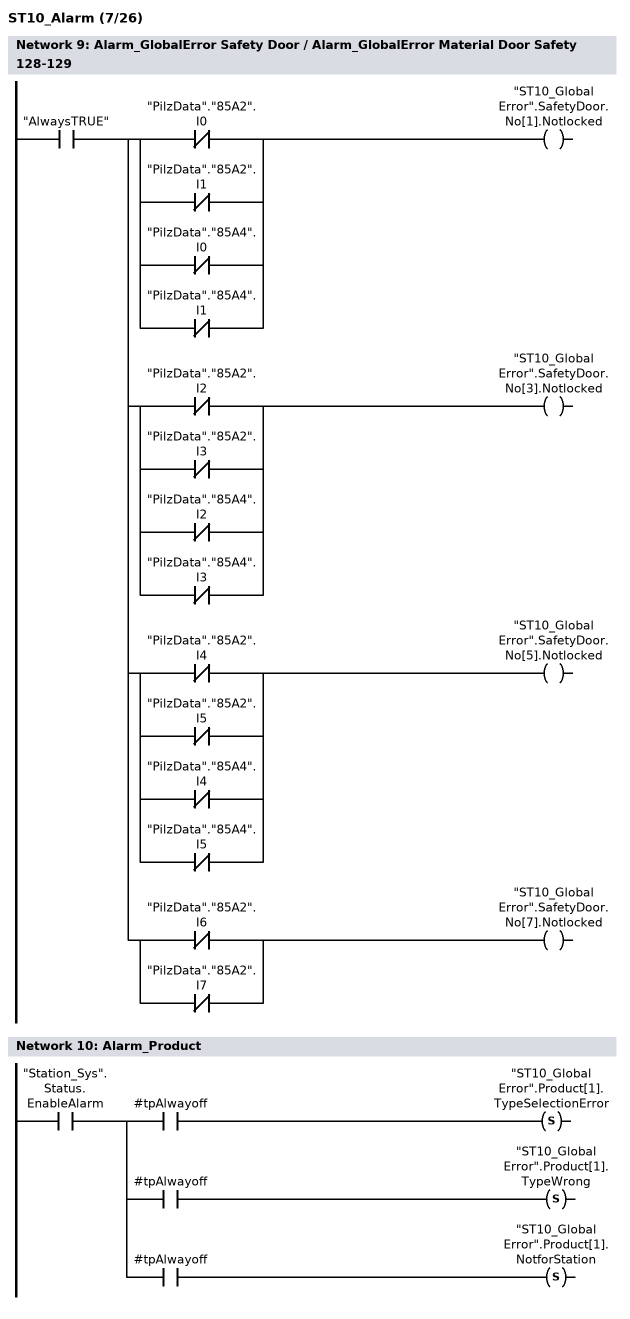
   RUNG wire#powerrail
      Contact( "AlwaysTRUE" )
      wire#w1
      I_Contact( "PilzData"."85A2".I0 )
      wire#w2
      Coil( "ST10_GlobalError".SafetyDoor.No[1].Notlocked )
   END_RUNG
   RUNG wire#w1
      I_Contact( "PilzData"."85A2".I1 )
   END_RUNG wire#w2
   RUNG wire#w1
      I_Contact( "PilzData"."85A4".I0 )
   END_RUNG wire#w2
   RUNG wire#w1
      I_Contact( "PilzData"."85A4".I1 )
   END_RUNG wire#w2
   RUNG wire#w1
      I_Contact( "PilzData"."85A2".I2 )
      wire#w3
      Coil( "ST10_GlobalError".SafetyDoor.No[3].Notlocked )
   END_RUNG
   RUNG wire#w1
      I_Contact( "PilzData"."85A2".I3 )
   END_RUNG wire#w3
   RUNG wire#w1
      I_Contact( "PilzData"."85A4".I2 )
   END_RUNG wire#w3
   RUNG wire#w1
      I_Contact( "PilzData"."85A4".I3 )
   END_RUNG wire#w3
   RUNG wire#w1
      I_Contact( "PilzData"."85A2".I4 )
      wire#w4
      Coil( "ST10_GlobalError".SafetyDoor.No[5].Notlocked )
   END_RUNG
   RUNG wire#w1
      I_Contact( "PilzData"."85A2".I5 )
   END_RUNG wire#w4
   RUNG wire#w1
      I_Contact( "PilzData"."85A4".I4 )
   END_RUNG wire#w4
   RUNG wire#w1
      I_Contact( "PilzData"."85A4".I5 )
   END_RUNG wire#w4
   RUNG wire#w1
      I_Contact( "PilzData"."85A2".I6 )
      wire#w5
      Coil( "ST10_GlobalError".SafetyDoor.No[7].Notlocked )
   END_RUNG
   RUNG wire#w1
      I_Contact( "PilzData"."85A2".I7 )
   END_RUNG wire#w5
   // the same network as SCL:
   "ST10_GlobalError".SafetyDoor.No[1].Notlocked := "AlwaysTRUE" AND (NOT "PilzData"."85A2".I0 OR NOT "PilzData"."85A2".I1 OR NOT "PilzData"."85A4".I0 OR NOT "PilzData"."85A4".I1);
   "ST10_GlobalError".SafetyDoor.No[3].Notlocked := "AlwaysTRUE" AND (NOT "PilzData"."85A2".I2 OR NOT "PilzData"."85A2".I3 OR NOT "PilzData"."85A4".I2 OR NOT "PilzData"."85A4".I3);
   "ST10_GlobalError".SafetyDoor.No[5].Notlocked := "AlwaysTRUE" AND (NOT "PilzData"."85A2".I4 OR NOT "PilzData"."85A2".I5 OR NOT "PilzData"."85A4".I4 OR NOT "PilzData"."85A4".I5);
   "ST10_GlobalError".SafetyDoor.No[7].Notlocked := "AlwaysTRUE" AND (NOT "PilzData"."85A2".I6 OR NOT "PilzData"."85A2".I7);
END_REGION

REGION Network 10: Alarm_Product
   RUNG wire#powerrail
      Contact( "Station_Sys".Status.EnableAlarm )
      wire#w1
      Contact( #tpAlwayoff )
      S_Coil( "ST10_GlobalError".Product[1].TypeSelectionError )
   END_RUNG
   RUNG wire#w1
      Contact( #tpAlwayoff )
      S_Coil( "ST10_GlobalError".Product[1].TypeWrong )
   END_RUNG
   RUNG wire#w1
      Contact( #tpAlwayoff )
      S_Coil( "ST10_GlobalError".Product[1].NotforStation )
   END_RUNG
   // the same network as SCL:
   IF "Station_Sys".Status.EnableAlarm AND #tpAlwayoff THEN
       "ST10_GlobalError".Product[1].TypeSelectionError := TRUE;
       "ST10_GlobalError".Product[1].TypeWrong := TRUE;
       "ST10_GlobalError".Product[1].NotforStation := TRUE;
   END_IF;
END_REGION

REGION Network 11 (SCL): Alarm_Fixture

   // IF "ST70_Sys".Status.EnableAlarm THEN

   //     //循环数量为工装检测的数量
   //     #FixtureNumber := 10;

   //     FOR #i := 1 TO #FixtureNumber DO
   //         "ST70_GlobalError".Fixture[#i].TypeError := NOT "ST70_GeneralData".FixtureIDCheck[#i].FixtureCheckResult;
   //     END_FOR;

   //     "ST70_GlobalError".Fixture[1].TypeError := NOT "ST70_GeneralData".FixtureIDCheck[11].FixtureCheckResult;
   //     "ST70_GlobalError".Fixture[2].TypeError := NOT "ST70_GeneralData".FixtureIDCheck[12].FixtureCheckResult;
   // END_IF;
END_REGION

REGION Network 12: ------------------------------------------------ A ---------------------------------------------------
END_REGION

REGION Network 13: ALightCuritTouch
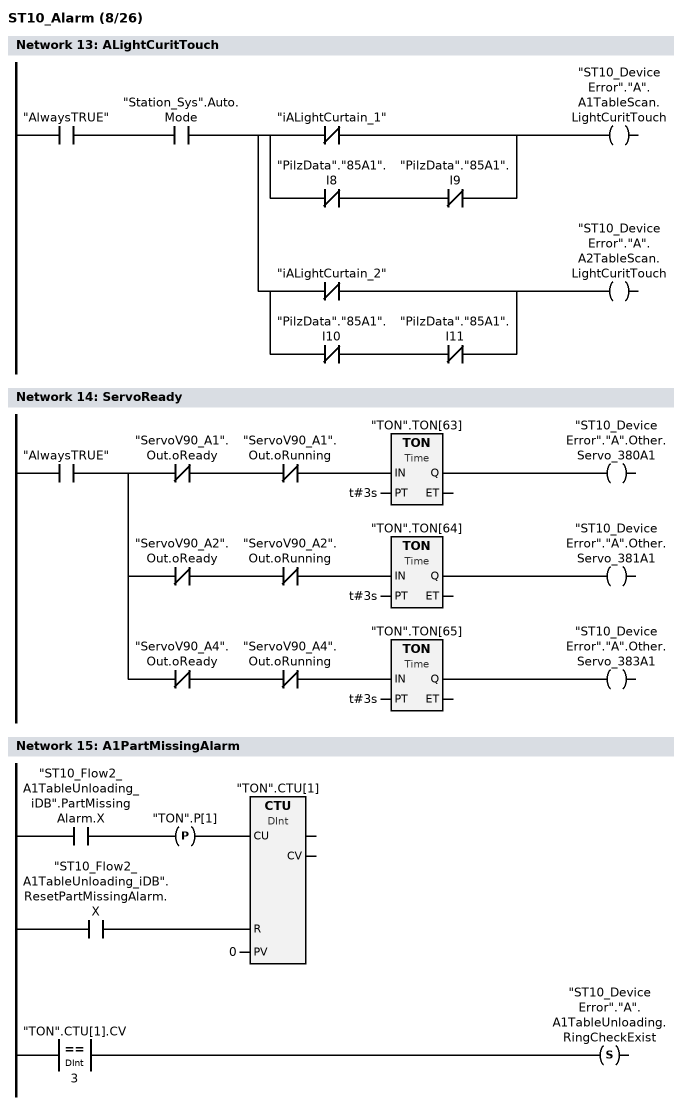
   RUNG wire#powerrail
      Contact( "AlwaysTRUE" )
      Contact( "Station_Sys".Auto.Mode )
      wire#w1
      I_Contact( "iALightCurtain_1" )
      wire#w2
      Coil( "ST10_DeviceError"."A".A1TableScan.LightCuritTouch )
   END_RUNG
   RUNG wire#w1
      I_Contact( "PilzData"."85A1".I8 )
      I_Contact( "PilzData"."85A1".I9 )
   END_RUNG wire#w2
   RUNG wire#w1
      I_Contact( "iALightCurtain_2" )
      wire#w3
      Coil( "ST10_DeviceError"."A".A2TableScan.LightCuritTouch )
   END_RUNG
   RUNG wire#w1
      I_Contact( "PilzData"."85A1".I10 )
      I_Contact( "PilzData"."85A1".I11 )
   END_RUNG wire#w3
   // the same network as SCL:
   #_w1 := "AlwaysTRUE" AND "Station_Sys".Auto.Mode;
   "ST10_DeviceError"."A".A1TableScan.LightCuritTouch := #_w1 AND (NOT "iALightCurtain_1" OR (NOT "PilzData"."85A1".I8 AND NOT "PilzData"."85A1".I9));
   "ST10_DeviceError"."A".A2TableScan.LightCuritTouch := #_w1 AND (NOT "iALightCurtain_2" OR (NOT "PilzData"."85A1".I10 AND NOT "PilzData"."85A1".I11));
END_REGION

REGION Network 14: ServoReady
   RUNG wire#powerrail
      Contact( "AlwaysTRUE" )
      wire#w1
      I_Contact( "ServoV90_A1".Out.oReady )
      I_Contact( "ServoV90_A1".Out.oRunning )
      { S7_Templates := "time_type := Time" } "TON".TON[63].TON(pt := t#3s, et =>)
      Coil( "ST10_DeviceError"."A".Other.Servo_380A1 )
   END_RUNG
   RUNG wire#w1
      I_Contact( "ServoV90_A2".Out.oReady )
      I_Contact( "ServoV90_A2".Out.oRunning )
      { S7_Templates := "time_type := Time" } "TON".TON[64].TON(pt := t#3s, et =>)
      Coil( "ST10_DeviceError"."A".Other.Servo_381A1 )
   END_RUNG
   RUNG wire#w1
      I_Contact( "ServoV90_A4".Out.oReady )
      I_Contact( "ServoV90_A4".Out.oRunning )
      { S7_Templates := "time_type := Time" } "TON".TON[65].TON(pt := t#3s, et =>)
      Coil( "ST10_DeviceError"."A".Other.Servo_383A1 )
   END_RUNG
   // the same network as SCL:
   "TON".TON[63].TON(IN := "AlwaysTRUE" AND NOT "ServoV90_A1".Out.oReady AND NOT "ServoV90_A1".Out.oRunning,
                     PT := t#3s);
   "ST10_DeviceError"."A".Other.Servo_380A1 := "TON".TON[63].Q;
   "TON".TON[64].TON(IN := "AlwaysTRUE" AND NOT "ServoV90_A2".Out.oReady AND NOT "ServoV90_A2".Out.oRunning,
                     PT := t#3s);
   "ST10_DeviceError"."A".Other.Servo_381A1 := "TON".TON[64].Q;
   "TON".TON[65].TON(IN := "AlwaysTRUE" AND NOT "ServoV90_A4".Out.oReady AND NOT "ServoV90_A4".Out.oRunning,
                     PT := t#3s);
   "ST10_DeviceError"."A".Other.Servo_383A1 := "TON".TON[65].Q;
END_REGION

REGION Network 15: A1PartMissingAlarm
   RUNG wire#powerrail
      Contact( "ST10_Flow2_A1TableUnloading_iDB".PartMissingAlarm.X )
      P_Trig( "TON".P[1] )
      { S7_Templates := "value_type := DInt" } "TON".CTU[1].CTU(r := wire#w1, pv := 0, cv =>)
   END_RUNG
   RUNG wire#powerrail
      Contact( "ST10_Flow2_A1TableUnloading_iDB".ResetPartMissingAlarm.X )
   END_RUNG wire#w1
   RUNG wire#powerrail
      { S7_Templates := "SrcType := DInt" } EQ_Contact(in1 := "TON".CTU[1].CV, in2 := 3)
      S_Coil( "ST10_DeviceError"."A".A1TableUnloading.RingCheckExist )
   END_RUNG
   // the same network as SCL:
   #_w1 := "ST10_Flow2_A1TableUnloading_iDB".PartMissingAlarm.X AND NOT "TON".P[1];   // rising edge
   "TON".P[1] := "ST10_Flow2_A1TableUnloading_iDB".PartMissingAlarm.X;
   "TON".CTU[1].CTU(CU := #_w1, R := "ST10_Flow2_A1TableUnloading_iDB".ResetPartMissingAlarm.X, PV := 0);
   IF "TON".CTU[1].CV = 3 THEN "ST10_DeviceError"."A".A1TableUnloading.RingCheckExist := TRUE; END_IF;
END_REGION

REGION Network 16: A2PartMissingAlarm
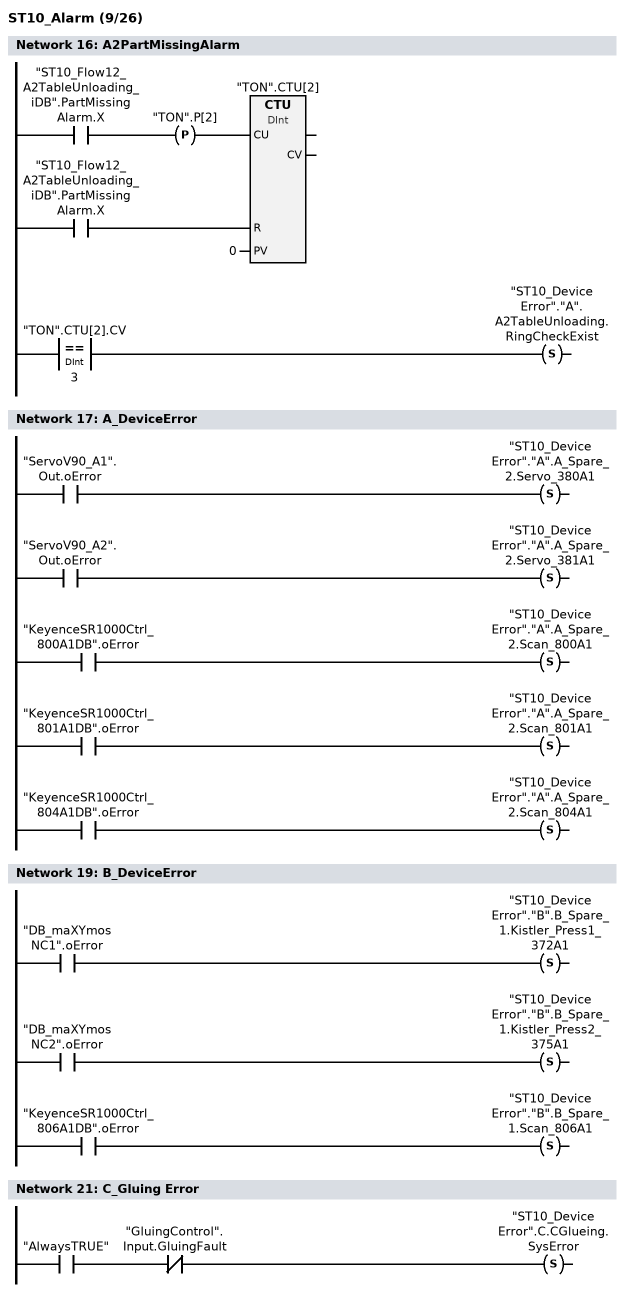
   RUNG wire#powerrail
      Contact( "ST10_Flow12_A2TableUnloading_iDB".PartMissingAlarm.X )
      P_Trig( "TON".P[2] )
      { S7_Templates := "value_type := DInt" } "TON".CTU[2].CTU(r := wire#w1, pv := 0, cv =>)
   END_RUNG
   RUNG wire#powerrail
      Contact( "ST10_Flow12_A2TableUnloading_iDB".PartMissingAlarm.X )
   END_RUNG wire#w1
   RUNG wire#powerrail
      { S7_Templates := "SrcType := DInt" } EQ_Contact(in1 := "TON".CTU[2].CV, in2 := 3)
      S_Coil( "ST10_DeviceError"."A".A2TableUnloading.RingCheckExist )
   END_RUNG
   // the same network as SCL:
   #_w1 := "ST10_Flow12_A2TableUnloading_iDB".PartMissingAlarm.X AND NOT "TON".P[2];   // rising edge
   "TON".P[2] := "ST10_Flow12_A2TableUnloading_iDB".PartMissingAlarm.X;
   "TON".CTU[2].CTU(CU := #_w1, R := "ST10_Flow12_A2TableUnloading_iDB".PartMissingAlarm.X, PV := 0);
   IF "TON".CTU[2].CV = 3 THEN "ST10_DeviceError"."A".A2TableUnloading.RingCheckExist := TRUE; END_IF;
END_REGION

REGION Network 17: A_DeviceError
   RUNG wire#powerrail
      Contact( "ServoV90_A1".Out.oError )
      S_Coil( "ST10_DeviceError"."A".A_Spare_2.Servo_380A1 )
   END_RUNG
   RUNG wire#powerrail
      Contact( "ServoV90_A2".Out.oError )
      S_Coil( "ST10_DeviceError"."A".A_Spare_2.Servo_381A1 )
   END_RUNG
   RUNG wire#powerrail
      Contact( "KeyenceSR1000Ctrl_800A1DB".oError )
      S_Coil( "ST10_DeviceError"."A".A_Spare_2.Scan_800A1 )
   END_RUNG
   RUNG wire#powerrail
      Contact( "KeyenceSR1000Ctrl_801A1DB".oError )
      S_Coil( "ST10_DeviceError"."A".A_Spare_2.Scan_801A1 )
   END_RUNG
   RUNG wire#powerrail
      Contact( "KeyenceSR1000Ctrl_804A1DB".oError )
      S_Coil( "ST10_DeviceError"."A".A_Spare_2.Scan_804A1 )
   END_RUNG
   // the same network as SCL:
   IF "ServoV90_A1".Out.oError THEN "ST10_DeviceError"."A".A_Spare_2.Servo_380A1 := TRUE; END_IF;
   IF "ServoV90_A2".Out.oError THEN "ST10_DeviceError"."A".A_Spare_2.Servo_381A1 := TRUE; END_IF;
   IF "KeyenceSR1000Ctrl_800A1DB".oError THEN "ST10_DeviceError"."A".A_Spare_2.Scan_800A1 := TRUE; END_IF;
   IF "KeyenceSR1000Ctrl_801A1DB".oError THEN "ST10_DeviceError"."A".A_Spare_2.Scan_801A1 := TRUE; END_IF;
   IF "KeyenceSR1000Ctrl_804A1DB".oError THEN "ST10_DeviceError"."A".A_Spare_2.Scan_804A1 := TRUE; END_IF;
END_REGION

REGION Network 18: ------------------------------------------------ B ---------------------------------------------------
END_REGION

REGION Network 19: B_DeviceError
   RUNG wire#powerrail
      Contact( "DB_maXYmosNC1".oError )
      S_Coil( "ST10_DeviceError"."B".B_Spare_1.Kistler_Press1_372A1 )
   END_RUNG
   RUNG wire#powerrail
      Contact( "DB_maXYmosNC2".oError )
      S_Coil( "ST10_DeviceError"."B".B_Spare_1.Kistler_Press2_375A1 )
   END_RUNG
   RUNG wire#powerrail
      Contact( "KeyenceSR1000Ctrl_806A1DB".oError )
      S_Coil( "ST10_DeviceError"."B".B_Spare_1.Scan_806A1 )
   END_RUNG
   // the same network as SCL:
   IF "DB_maXYmosNC1".oError THEN "ST10_DeviceError"."B".B_Spare_1.Kistler_Press1_372A1 := TRUE; END_IF;
   IF "DB_maXYmosNC2".oError THEN "ST10_DeviceError"."B".B_Spare_1.Kistler_Press2_375A1 := TRUE; END_IF;
   IF "KeyenceSR1000Ctrl_806A1DB".oError THEN "ST10_DeviceError"."B".B_Spare_1.Scan_806A1 := TRUE; END_IF;
END_REGION

REGION Network 20: ------------------------------------------------ C ---------------------------------------------------
END_REGION

REGION Network 21: C_Gluing Error
   RUNG wire#powerrail
      Contact( "AlwaysTRUE" )
      I_Contact( "GluingControl".Input.GluingFault )
      S_Coil( "ST10_DeviceError".C.CGlueing.SysError )
   END_RUNG
   // the same network as SCL:
   IF "AlwaysTRUE" AND NOT "GluingControl".Input.GluingFault THEN
       "ST10_DeviceError".C.CGlueing.SysError := TRUE;
   END_IF;
END_REGION

REGION Network 22: ServoReady
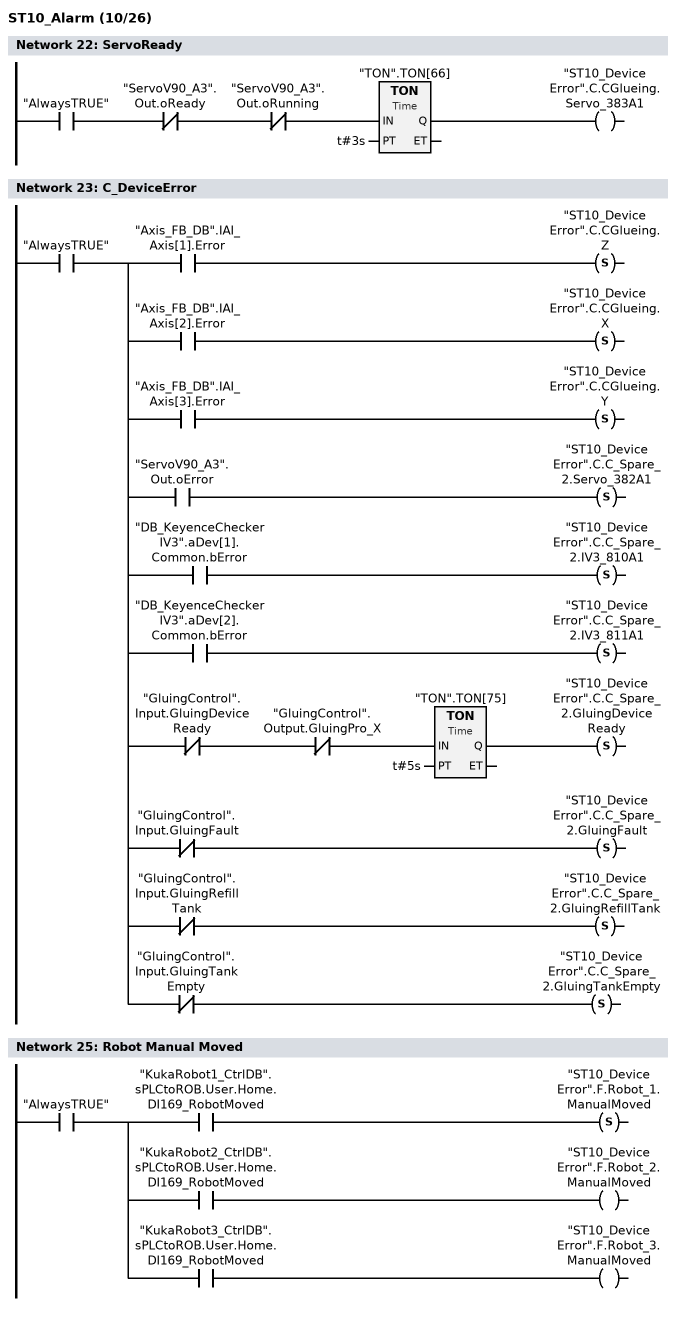
   RUNG wire#powerrail
      Contact( "AlwaysTRUE" )
      I_Contact( "ServoV90_A3".Out.oReady )
      I_Contact( "ServoV90_A3".Out.oRunning )
      { S7_Templates := "time_type := Time" } "TON".TON[66].TON(pt := t#3s, et =>)
      Coil( "ST10_DeviceError".C.CGlueing.Servo_383A1 )
   END_RUNG
   // the same network as SCL:
   "TON".TON[66].TON(IN := "AlwaysTRUE" AND NOT "ServoV90_A3".Out.oReady AND NOT "ServoV90_A3".Out.oRunning,
                     PT := t#3s);
   "ST10_DeviceError".C.CGlueing.Servo_383A1 := "TON".TON[66].Q;
END_REGION

REGION Network 23: C_DeviceError
   RUNG wire#powerrail
      Contact( "AlwaysTRUE" )
      wire#w1
      Contact( "Axis_FB_DB".IAI_Axis[1].Error )
      S_Coil( "ST10_DeviceError".C.CGlueing.Z )
   END_RUNG
   RUNG wire#w1
      Contact( "Axis_FB_DB".IAI_Axis[2].Error )
      S_Coil( "ST10_DeviceError".C.CGlueing.X )
   END_RUNG
   RUNG wire#w1
      Contact( "Axis_FB_DB".IAI_Axis[3].Error )
      S_Coil( "ST10_DeviceError".C.CGlueing.Y )
   END_RUNG
   RUNG wire#w1
      Contact( "ServoV90_A3".Out.oError )
      S_Coil( "ST10_DeviceError".C.C_Spare_2.Servo_382A1 )
   END_RUNG
   RUNG wire#w1
      Contact( "DB_KeyenceCheckerIV3".aDev[1].Common.bError )
      S_Coil( "ST10_DeviceError".C.C_Spare_2.IV3_810A1 )
   END_RUNG
   RUNG wire#w1
      Contact( "DB_KeyenceCheckerIV3".aDev[2].Common.bError )
      S_Coil( "ST10_DeviceError".C.C_Spare_2.IV3_811A1 )
   END_RUNG
   RUNG wire#w1
      I_Contact( "GluingControl".Input.GluingDeviceReady )
      I_Contact( "GluingControl".Output.GluingPro_X )
      { S7_Templates := "time_type := Time" } "TON".TON[75].TON(pt := t#5s, et =>)
      S_Coil( "ST10_DeviceError".C.C_Spare_2.GluingDeviceReady )
   END_RUNG
   RUNG wire#w1
      I_Contact( "GluingControl".Input.GluingFault )
      S_Coil( "ST10_DeviceError".C.C_Spare_2.GluingFault )
   END_RUNG
   RUNG wire#w1
      I_Contact( "GluingControl".Input.GluingRefillTank )
      S_Coil( "ST10_DeviceError".C.C_Spare_2.GluingRefillTank )
   END_RUNG
   RUNG wire#w1
      I_Contact( "GluingControl".Input.GluingTankEmpty )
      S_Coil( "ST10_DeviceError".C.C_Spare_2.GluingTankEmpty )
   END_RUNG
   // the same network as SCL:
   IF "AlwaysTRUE" AND "Axis_FB_DB".IAI_Axis[1].Error THEN "ST10_DeviceError".C.CGlueing.Z := TRUE; END_IF;
   IF "AlwaysTRUE" AND "Axis_FB_DB".IAI_Axis[2].Error THEN "ST10_DeviceError".C.CGlueing.X := TRUE; END_IF;
   IF "AlwaysTRUE" AND "Axis_FB_DB".IAI_Axis[3].Error THEN "ST10_DeviceError".C.CGlueing.Y := TRUE; END_IF;
   IF "AlwaysTRUE" AND "ServoV90_A3".Out.oError THEN
       "ST10_DeviceError".C.C_Spare_2.Servo_382A1 := TRUE;
   END_IF;
   IF "AlwaysTRUE" AND "DB_KeyenceCheckerIV3".aDev[1].Common.bError THEN
       "ST10_DeviceError".C.C_Spare_2.IV3_810A1 := TRUE;
   END_IF;
   IF "AlwaysTRUE" AND "DB_KeyenceCheckerIV3".aDev[2].Common.bError THEN
       "ST10_DeviceError".C.C_Spare_2.IV3_811A1 := TRUE;
   END_IF;
   "TON".TON[75].TON(IN := "AlwaysTRUE" AND NOT "GluingControl".Input.GluingDeviceReady AND NOT "GluingControl".Output.GluingPro_X,
                     PT := t#5s);
   IF "TON".TON[75].Q THEN "ST10_DeviceError".C.C_Spare_2.GluingDeviceReady := TRUE; END_IF;
   IF "AlwaysTRUE" AND NOT "GluingControl".Input.GluingFault THEN
       "ST10_DeviceError".C.C_Spare_2.GluingFault := TRUE;
   END_IF;
   IF "AlwaysTRUE" AND NOT "GluingControl".Input.GluingRefillTank THEN
       "ST10_DeviceError".C.C_Spare_2.GluingRefillTank := TRUE;
   END_IF;
   IF "AlwaysTRUE" AND NOT "GluingControl".Input.GluingTankEmpty THEN
       "ST10_DeviceError".C.C_Spare_2.GluingTankEmpty := TRUE;
   END_IF;
END_REGION

REGION Network 24: ------------------------------------------------ F ---------------------------------------------------
END_REGION

REGION Network 25: Robot Manual Moved
   RUNG wire#powerrail
      Contact( "AlwaysTRUE" )
      wire#w1
      Contact( "KukaRobot1_CtrlDB".sPLCtoROB.User.Home.DI169_RobotMoved )
      S_Coil( "ST10_DeviceError".F.Robot_1.ManualMoved )
   END_RUNG
   RUNG wire#w1
      Contact( "KukaRobot2_CtrlDB".sPLCtoROB.User.Home.DI169_RobotMoved )
      Coil( "ST10_DeviceError".F.Robot_2.ManualMoved )
   END_RUNG
   RUNG wire#w1
      Contact( "KukaRobot3_CtrlDB".sPLCtoROB.User.Home.DI169_RobotMoved )
      Coil( "ST10_DeviceError".F.Robot_3.ManualMoved )
   END_RUNG
   // the same network as SCL:
   IF "AlwaysTRUE" AND "KukaRobot1_CtrlDB".sPLCtoROB.User.Home.DI169_RobotMoved THEN
       "ST10_DeviceError".F.Robot_1.ManualMoved := TRUE;
   END_IF;
   "ST10_DeviceError".F.Robot_2.ManualMoved := "AlwaysTRUE" AND "KukaRobot2_CtrlDB".sPLCtoROB.User.Home.DI169_RobotMoved;
   "ST10_DeviceError".F.Robot_3.ManualMoved := "AlwaysTRUE" AND "KukaRobot3_CtrlDB".sPLCtoROB.User.Home.DI169_RobotMoved;
END_REGION

REGION Network 26: Robot 1 Not auto Mode
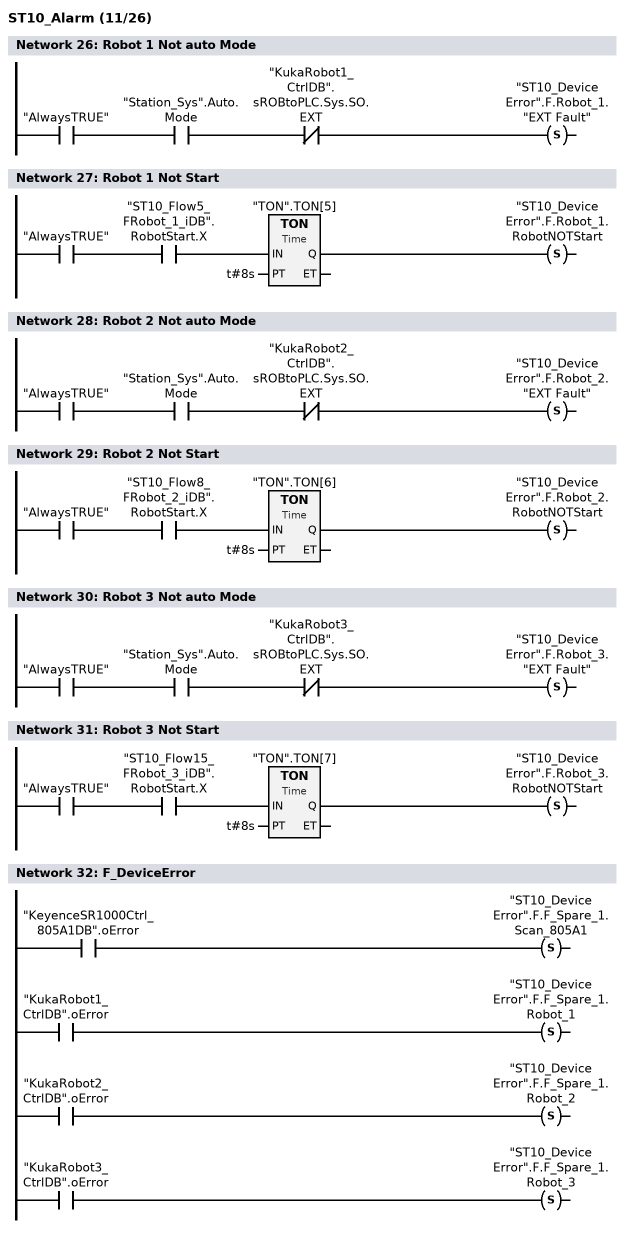
   RUNG wire#powerrail
      Contact( "AlwaysTRUE" )
      Contact( "Station_Sys".Auto.Mode )
      I_Contact( "KukaRobot1_CtrlDB".sROBtoPLC.Sys.SO.EXT )
      S_Coil( "ST10_DeviceError".F.Robot_1."EXT Fault" )
   END_RUNG
   // the same network as SCL:
   IF "AlwaysTRUE" AND "Station_Sys".Auto.Mode AND NOT "KukaRobot1_CtrlDB".sROBtoPLC.Sys.SO.EXT THEN
       "ST10_DeviceError".F.Robot_1."EXT Fault" := TRUE;
   END_IF;
END_REGION

REGION Network 27: Robot 1 Not Start
   RUNG wire#powerrail
      Contact( "AlwaysTRUE" )
      Contact( "ST10_Flow5_FRobot_1_iDB".RobotStart.X )
      { S7_Templates := "time_type := Time" } "TON".TON[5].TON(pt := t#8s, et =>)
      S_Coil( "ST10_DeviceError".F.Robot_1.RobotNOTStart )
   END_RUNG
   // the same network as SCL:
   "TON".TON[5].TON(IN := "AlwaysTRUE" AND "ST10_Flow5_FRobot_1_iDB".RobotStart.X, PT := t#8s);
   IF "TON".TON[5].Q THEN "ST10_DeviceError".F.Robot_1.RobotNOTStart := TRUE; END_IF;
END_REGION

REGION Network 28: Robot 2 Not auto Mode
   RUNG wire#powerrail
      Contact( "AlwaysTRUE" )
      Contact( "Station_Sys".Auto.Mode )
      I_Contact( "KukaRobot2_CtrlDB".sROBtoPLC.Sys.SO.EXT )
      S_Coil( "ST10_DeviceError".F.Robot_2."EXT Fault" )
   END_RUNG
   // the same network as SCL:
   IF "AlwaysTRUE" AND "Station_Sys".Auto.Mode AND NOT "KukaRobot2_CtrlDB".sROBtoPLC.Sys.SO.EXT THEN
       "ST10_DeviceError".F.Robot_2."EXT Fault" := TRUE;
   END_IF;
END_REGION

REGION Network 29: Robot 2 Not Start
   RUNG wire#powerrail
      Contact( "AlwaysTRUE" )
      Contact( "ST10_Flow8_FRobot_2_iDB".RobotStart.X )
      { S7_Templates := "time_type := Time" } "TON".TON[6].TON(pt := t#8s, et =>)
      S_Coil( "ST10_DeviceError".F.Robot_2.RobotNOTStart )
   END_RUNG
   // the same network as SCL:
   "TON".TON[6].TON(IN := "AlwaysTRUE" AND "ST10_Flow8_FRobot_2_iDB".RobotStart.X, PT := t#8s);
   IF "TON".TON[6].Q THEN "ST10_DeviceError".F.Robot_2.RobotNOTStart := TRUE; END_IF;
END_REGION

REGION Network 30: Robot 3 Not auto Mode
   RUNG wire#powerrail
      Contact( "AlwaysTRUE" )
      Contact( "Station_Sys".Auto.Mode )
      I_Contact( "KukaRobot3_CtrlDB".sROBtoPLC.Sys.SO.EXT )
      S_Coil( "ST10_DeviceError".F.Robot_3."EXT Fault" )
   END_RUNG
   // the same network as SCL:
   IF "AlwaysTRUE" AND "Station_Sys".Auto.Mode AND NOT "KukaRobot3_CtrlDB".sROBtoPLC.Sys.SO.EXT THEN
       "ST10_DeviceError".F.Robot_3."EXT Fault" := TRUE;
   END_IF;
END_REGION

REGION Network 31: Robot 3 Not Start
   RUNG wire#powerrail
      Contact( "AlwaysTRUE" )
      Contact( "ST10_Flow15_FRobot_3_iDB".RobotStart.X )
      { S7_Templates := "time_type := Time" } "TON".TON[7].TON(pt := t#8s, et =>)
      S_Coil( "ST10_DeviceError".F.Robot_3.RobotNOTStart )
   END_RUNG
   // the same network as SCL:
   "TON".TON[7].TON(IN := "AlwaysTRUE" AND "ST10_Flow15_FRobot_3_iDB".RobotStart.X, PT := t#8s);
   IF "TON".TON[7].Q THEN "ST10_DeviceError".F.Robot_3.RobotNOTStart := TRUE; END_IF;
END_REGION

REGION Network 32: F_DeviceError
   RUNG wire#powerrail
      Contact( "KeyenceSR1000Ctrl_805A1DB".oError )
      S_Coil( "ST10_DeviceError".F.F_Spare_1.Scan_805A1 )
   END_RUNG
   RUNG wire#powerrail
      Contact( "KukaRobot1_CtrlDB".oError )
      S_Coil( "ST10_DeviceError".F.F_Spare_1.Robot_1 )
   END_RUNG
   RUNG wire#powerrail
      Contact( "KukaRobot2_CtrlDB".oError )
      S_Coil( "ST10_DeviceError".F.F_Spare_1.Robot_2 )
   END_RUNG
   RUNG wire#powerrail
      Contact( "KukaRobot3_CtrlDB".oError )
      S_Coil( "ST10_DeviceError".F.F_Spare_1.Robot_3 )
   END_RUNG
   // the same network as SCL:
   IF "KeyenceSR1000Ctrl_805A1DB".oError THEN "ST10_DeviceError".F.F_Spare_1.Scan_805A1 := TRUE; END_IF;
   IF "KukaRobot1_CtrlDB".oError THEN "ST10_DeviceError".F.F_Spare_1.Robot_1 := TRUE; END_IF;
   IF "KukaRobot2_CtrlDB".oError THEN "ST10_DeviceError".F.F_Spare_1.Robot_2 := TRUE; END_IF;
   IF "KukaRobot3_CtrlDB".oError THEN "ST10_DeviceError".F.F_Spare_1.Robot_3 := TRUE; END_IF;
END_REGION

REGION Network 33: ------------------------------------------------ H ---------------------------------------------------
END_REGION

REGION Network 34: F_DeviceError
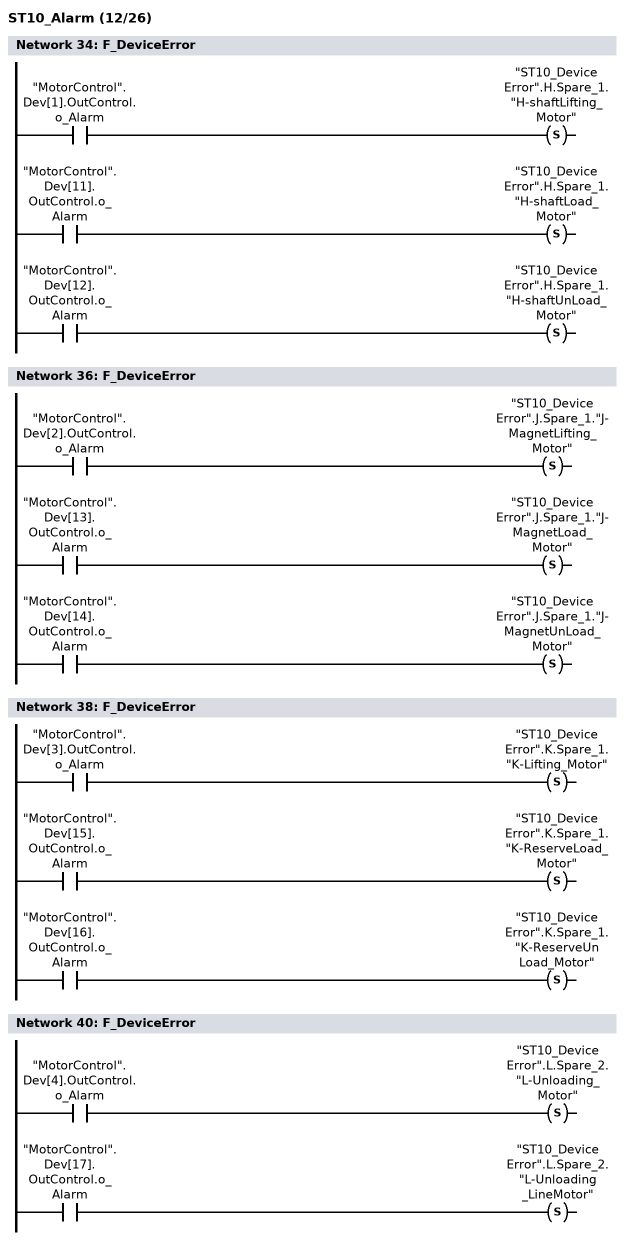
   RUNG wire#powerrail
      Contact( "MotorControl".Dev[1].OutControl.o_Alarm )
      S_Coil( "ST10_DeviceError".H.Spare_1."H-shaftLifting_Motor" )
   END_RUNG
   RUNG wire#powerrail
      Contact( "MotorControl".Dev[11].OutControl.o_Alarm )
      S_Coil( "ST10_DeviceError".H.Spare_1."H-shaftLoad_Motor" )
   END_RUNG
   RUNG wire#powerrail
      Contact( "MotorControl".Dev[12].OutControl.o_Alarm )
      S_Coil( "ST10_DeviceError".H.Spare_1."H-shaftUnLoad_Motor" )
   END_RUNG
   // the same network as SCL:
   IF "MotorControl".Dev[1].OutControl.o_Alarm THEN
       "ST10_DeviceError".H.Spare_1."H-shaftLifting_Motor" := TRUE;
   END_IF;
   IF "MotorControl".Dev[11].OutControl.o_Alarm THEN
       "ST10_DeviceError".H.Spare_1."H-shaftLoad_Motor" := TRUE;
   END_IF;
   IF "MotorControl".Dev[12].OutControl.o_Alarm THEN
       "ST10_DeviceError".H.Spare_1."H-shaftUnLoad_Motor" := TRUE;
   END_IF;
END_REGION

REGION Network 35: ------------------------------------------------ J ---------------------------------------------------
END_REGION

REGION Network 36: F_DeviceError
   RUNG wire#powerrail
      Contact( "MotorControl".Dev[2].OutControl.o_Alarm )
      S_Coil( "ST10_DeviceError".J.Spare_1."J-MagnetLifting_Motor" )
   END_RUNG
   RUNG wire#powerrail
      Contact( "MotorControl".Dev[13].OutControl.o_Alarm )
      S_Coil( "ST10_DeviceError".J.Spare_1."J-MagnetLoad_Motor" )
   END_RUNG
   RUNG wire#powerrail
      Contact( "MotorControl".Dev[14].OutControl.o_Alarm )
      S_Coil( "ST10_DeviceError".J.Spare_1."J-MagnetUnLoad_Motor" )
   END_RUNG
   // the same network as SCL:
   IF "MotorControl".Dev[2].OutControl.o_Alarm THEN
       "ST10_DeviceError".J.Spare_1."J-MagnetLifting_Motor" := TRUE;
   END_IF;
   IF "MotorControl".Dev[13].OutControl.o_Alarm THEN
       "ST10_DeviceError".J.Spare_1."J-MagnetLoad_Motor" := TRUE;
   END_IF;
   IF "MotorControl".Dev[14].OutControl.o_Alarm THEN
       "ST10_DeviceError".J.Spare_1."J-MagnetUnLoad_Motor" := TRUE;
   END_IF;
END_REGION

REGION Network 37: ------------------------------------------------ K ---------------------------------------------------
END_REGION

REGION Network 38: F_DeviceError
   RUNG wire#powerrail
      Contact( "MotorControl".Dev[3].OutControl.o_Alarm )
      S_Coil( "ST10_DeviceError".K.Spare_1."K-Lifting_Motor" )
   END_RUNG
   RUNG wire#powerrail
      Contact( "MotorControl".Dev[15].OutControl.o_Alarm )
      S_Coil( "ST10_DeviceError".K.Spare_1."K-ReserveLoad_Motor" )
   END_RUNG
   RUNG wire#powerrail
      Contact( "MotorControl".Dev[16].OutControl.o_Alarm )
      S_Coil( "ST10_DeviceError".K.Spare_1."K-ReserveUnLoad_Motor" )
   END_RUNG
   // the same network as SCL:
   IF "MotorControl".Dev[3].OutControl.o_Alarm THEN
       "ST10_DeviceError".K.Spare_1."K-Lifting_Motor" := TRUE;
   END_IF;
   IF "MotorControl".Dev[15].OutControl.o_Alarm THEN
       "ST10_DeviceError".K.Spare_1."K-ReserveLoad_Motor" := TRUE;
   END_IF;
   IF "MotorControl".Dev[16].OutControl.o_Alarm THEN
       "ST10_DeviceError".K.Spare_1."K-ReserveUnLoad_Motor" := TRUE;
   END_IF;
END_REGION

REGION Network 39: ------------------------------------------------ L ---------------------------------------------------
END_REGION

REGION Network 40: F_DeviceError
   RUNG wire#powerrail
      Contact( "MotorControl".Dev[4].OutControl.o_Alarm )
      S_Coil( "ST10_DeviceError".L.Spare_2."L-Unloading_Motor" )
   END_RUNG
   RUNG wire#powerrail
      Contact( "MotorControl".Dev[17].OutControl.o_Alarm )
      S_Coil( "ST10_DeviceError".L.Spare_2."L-Unloading _LineMotor" )
   END_RUNG
   // the same network as SCL:
   IF "MotorControl".Dev[4].OutControl.o_Alarm THEN
       "ST10_DeviceError".L.Spare_2."L-Unloading_Motor" := TRUE;
   END_IF;
   IF "MotorControl".Dev[17].OutControl.o_Alarm THEN
       "ST10_DeviceError".L.Spare_2."L-Unloading _LineMotor" := TRUE;
   END_IF;
END_REGION

REGION Network 41: Alarm_Breaker / 断路器
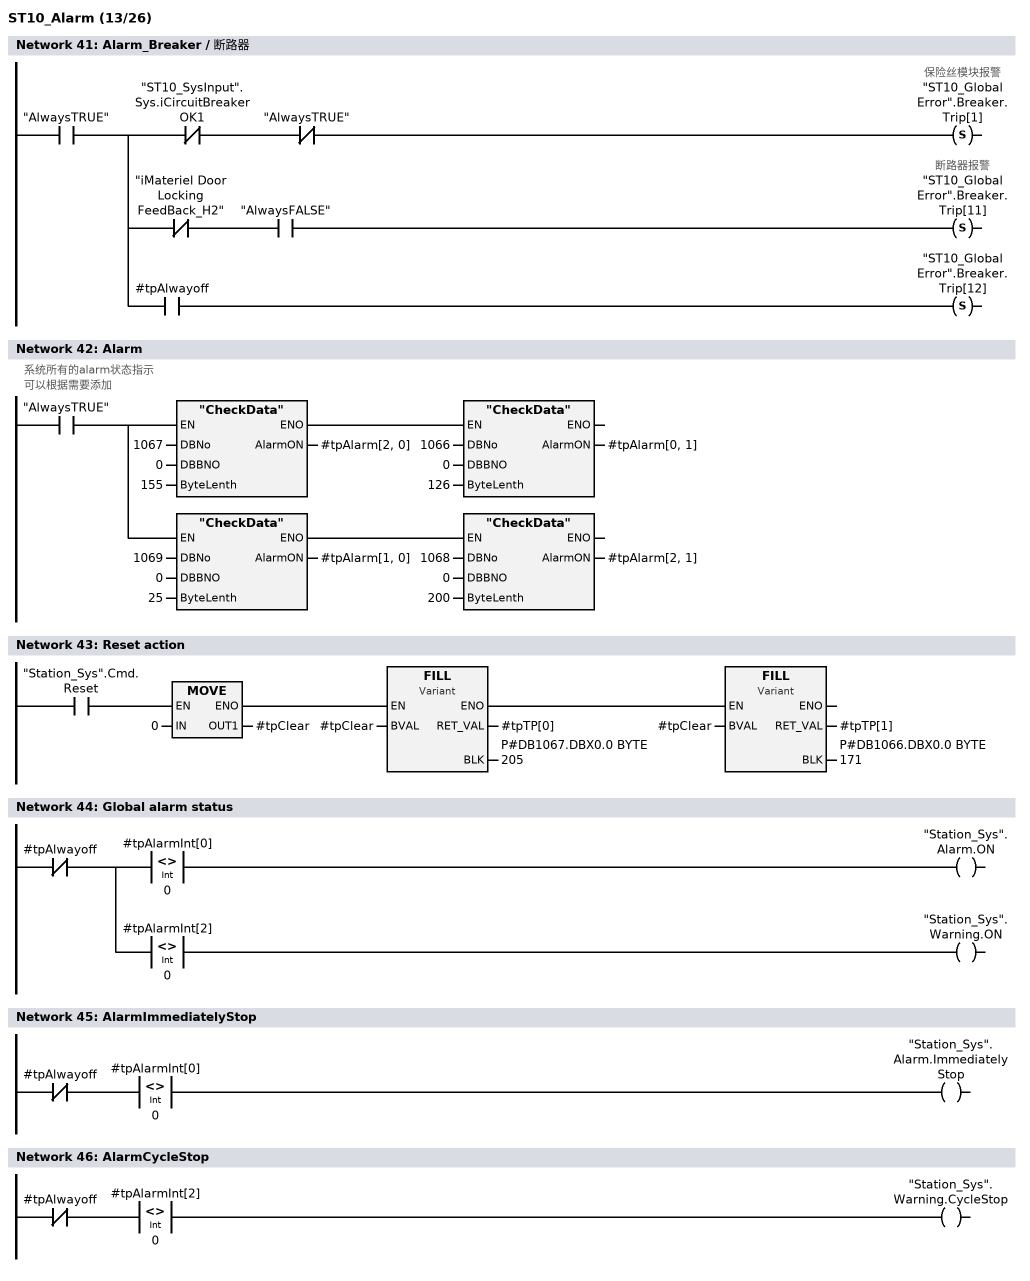
   RUNG wire#powerrail
      Contact( "AlwaysTRUE" )
      wire#w1
      I_Contact( "ST10_SysInput".Sys.iCircuitBreakerOK1 )
      I_Contact( "AlwaysTRUE" )
      S_Coil( "ST10_GlobalError".Breaker.Trip[1] )   // 保险丝模块报警
   END_RUNG
   RUNG wire#w1
      I_Contact( "iMateriel Door Locking FeedBack_H2" )
      Contact( "AlwaysFALSE" )
      S_Coil( "ST10_GlobalError".Breaker.Trip[11] )   // 断路器报警
   END_RUNG
   RUNG wire#w1
      Contact( #tpAlwayoff )
      S_Coil( "ST10_GlobalError".Breaker.Trip[12] )
   END_RUNG
   // the same network as SCL:
   IF "AlwaysTRUE" AND NOT "ST10_SysInput".Sys.iCircuitBreakerOK1 AND NOT "AlwaysTRUE" THEN
       "ST10_GlobalError".Breaker.Trip[1] := TRUE;   // 保险丝模块报警
   END_IF;
   IF "AlwaysTRUE" AND NOT "iMateriel Door Locking FeedBack_H2" AND "AlwaysFALSE" THEN
       "ST10_GlobalError".Breaker.Trip[11] := TRUE;   // 断路器报警
   END_IF;
   IF "AlwaysTRUE" AND #tpAlwayoff THEN "ST10_GlobalError".Breaker.Trip[12] := TRUE; END_IF;
END_REGION

REGION Network 42: Alarm
   // 系统所有的alarm状态指示
   // 可以根据需要添加
   RUNG wire#powerrail
      Contact( "AlwaysTRUE" )
      wire#w1
      "CheckData"(DBNo := 1067, DBBNO := 0, ByteLenth := 155, AlarmON => #tpAlarm[2, 0])
      "CheckData"(DBNo := 1066, DBBNO := 0, ByteLenth := 126, AlarmON => #tpAlarm[0, 1])
   END_RUNG
   RUNG wire#w1
      "CheckData"(DBNo := 1069, DBBNO := 0, ByteLenth := 25, AlarmON => #tpAlarm[1, 0])
      "CheckData"(DBNo := 1068, DBBNO := 0, ByteLenth := 200, AlarmON => #tpAlarm[2, 1])
   END_RUNG
   // the same network as SCL:
   #_w2 := "AlwaysTRUE";
   "CheckData"(EN := "AlwaysTRUE",
               DBNo := 1067,
               DBBNO := 0,
               ByteLenth := 155,
               AlarmON => #tpAlarm[2, 0],
               ENO => #_w1);
   IF #_w1 THEN "CheckData"(DBNo := 1066, DBBNO := 0, ByteLenth := 126, AlarmON => #tpAlarm[0, 1]); END_IF;
   "CheckData"(EN := #_w2, DBNo := 1069, DBBNO := 0, ByteLenth := 25, AlarmON => #tpAlarm[1, 0], ENO => #_w3);
   IF #_w3 THEN "CheckData"(DBNo := 1068, DBBNO := 0, ByteLenth := 200, AlarmON => #tpAlarm[2, 1]); END_IF;
END_REGION

REGION Network 43: Reset action
   RUNG wire#powerrail
      Contact( "Station_Sys".Cmd.Reset )
      Move(in := 0, out1 => #tpClear)
      { S7_Templates := "ptr_type := Variant" } FILL(BVAL := #tpClear, RET_VAL => #tpTP[0], BLK => P#DB1067.DBX0.0 BYTE 205)
      { S7_Templates := "ptr_type := Variant" } FILL(BVAL := #tpClear, RET_VAL => #tpTP[1], BLK => P#DB1066.DBX0.0 BYTE 171)
   END_RUNG
   // the same network as SCL:
   IF "Station_Sys".Cmd.Reset THEN #tpClear := 0; END_IF;
   #tpTP[0] := FILL(EN := "Station_Sys".Cmd.Reset,
                    BVAL := #tpClear,
                    BLK => P#DB1067.DBX0.0 BYTE 205,
                    ENO => #_w1);
   IF #_w1 THEN #tpTP[1] := FILL(BVAL := #tpClear, BLK => P#DB1066.DBX0.0 BYTE 171); END_IF;
END_REGION

REGION Network 44: Global alarm status
   RUNG wire#powerrail
      I_Contact( #tpAlwayoff )
      wire#w1
      { S7_Templates := "SrcType := Int" } NE_Contact(in1 := #tpAlarmInt[0], in2 := 0)
      Coil( "Station_Sys".Alarm.ON )
   END_RUNG
   RUNG wire#w1
      { S7_Templates := "SrcType := Int" } NE_Contact(in1 := #tpAlarmInt[2], in2 := 0)
      Coil( "Station_Sys".Warning.ON )
   END_RUNG
   // the same network as SCL:
   "Station_Sys".Alarm.ON := NOT #tpAlwayoff AND (#tpAlarmInt[0] <> 0);
   "Station_Sys".Warning.ON := NOT #tpAlwayoff AND (#tpAlarmInt[2] <> 0);
END_REGION

REGION Network 45: AlarmImmediatelyStop
   RUNG wire#powerrail
      I_Contact( #tpAlwayoff )
      { S7_Templates := "SrcType := Int" } NE_Contact(in1 := #tpAlarmInt[0], in2 := 0)
      Coil( "Station_Sys".Alarm.ImmediatelyStop )
   END_RUNG
   // the same network as SCL:
   "Station_Sys".Alarm.ImmediatelyStop := NOT #tpAlwayoff AND (#tpAlarmInt[0] <> 0);
END_REGION

REGION Network 46: AlarmCycleStop
   RUNG wire#powerrail
      I_Contact( #tpAlwayoff )
      { S7_Templates := "SrcType := Int" } NE_Contact(in1 := #tpAlarmInt[2], in2 := 0)
      Coil( "Station_Sys".Warning.CycleStop )
   END_RUNG
   // the same network as SCL:
   "Station_Sys".Warning.CycleStop := NOT #tpAlwayoff AND (#tpAlarmInt[2] <> 0);
END_REGION

REGION Network 47: -----------------------------------------------------------AlarmStatus----------------------------------------------------------------
END_REGION

REGION Network 48: ******************** H_Shaft loading ********************
END_REGION

REGION Network 49: H
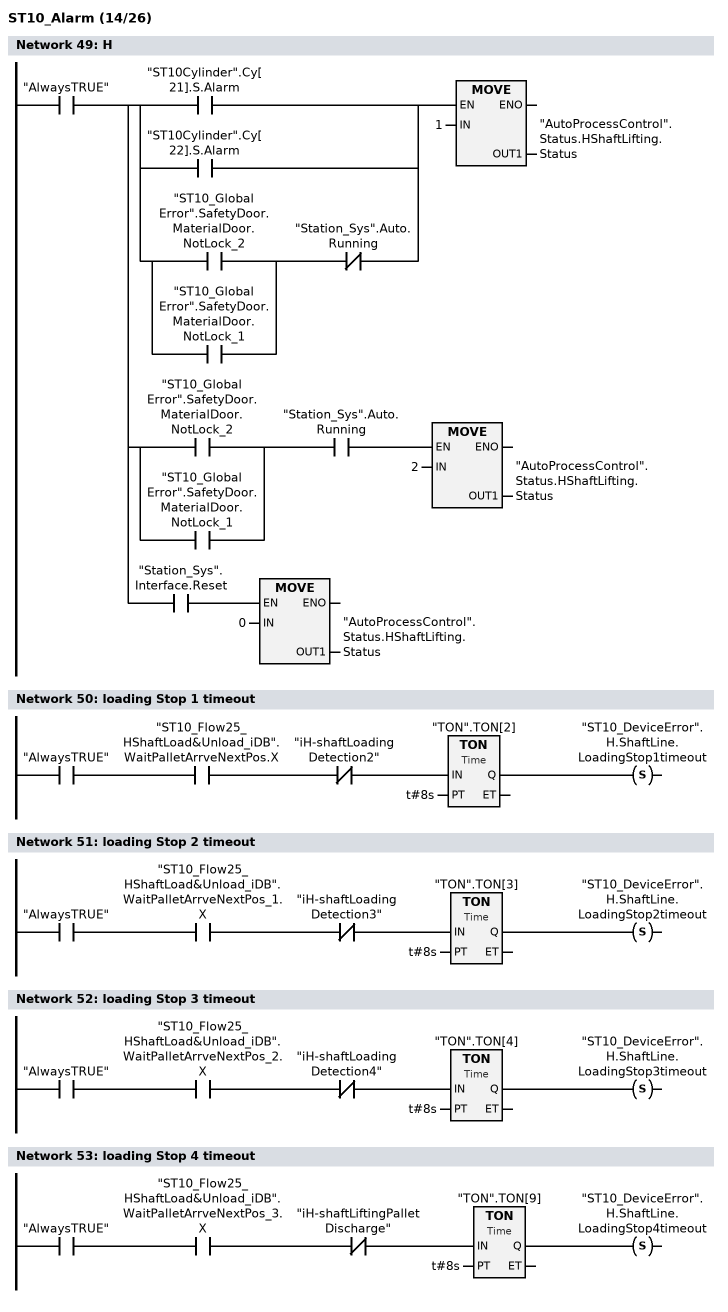
   RUNG wire#powerrail
      Contact( "AlwaysTRUE" )
      wire#w1
      Contact( "ST10Cylinder".Cy[21].S.Alarm )
      wire#w2
      Move(in := 1, out1 => "AutoProcessControl".Status.HShaftLifting.Status)
   END_RUNG
   RUNG wire#w1
      Contact( "ST10Cylinder".Cy[22].S.Alarm )
   END_RUNG wire#w2
   RUNG wire#w1
      Contact( "ST10_GlobalError".SafetyDoor.MaterialDoor.NotLock_2 )
      wire#w3
      I_Contact( "Station_Sys".Auto.Running )
   END_RUNG wire#w2
   RUNG wire#w1
      Contact( "ST10_GlobalError".SafetyDoor.MaterialDoor.NotLock_1 )
   END_RUNG wire#w3
   RUNG wire#w1
      Contact( "ST10_GlobalError".SafetyDoor.MaterialDoor.NotLock_2 )
      wire#w4
      Contact( "Station_Sys".Auto.Running )
      Move(in := 2, out1 => "AutoProcessControl".Status.HShaftLifting.Status)
   END_RUNG
   RUNG wire#w1
      Contact( "ST10_GlobalError".SafetyDoor.MaterialDoor.NotLock_1 )
   END_RUNG wire#w4
   RUNG wire#w1
      Contact( "Station_Sys".Interface.Reset )
      Move(in := 0, out1 => "AutoProcessControl".Status.HShaftLifting.Status)
   END_RUNG
   // the same network as SCL:
   IF "AlwaysTRUE" AND ("ST10Cylinder".Cy[21].S.Alarm OR "ST10Cylinder".Cy[22].S.Alarm OR (("ST10_GlobalError".SafetyDoor.MaterialDoor.NotLock_2 OR "ST10_GlobalError".SafetyDoor.MaterialDoor.NotLock_1) AND NOT "Station_Sys".Auto.Running)) THEN
       "AutoProcessControl".Status.HShaftLifting.Status := 1;
   END_IF;
   IF "AlwaysTRUE" AND ("ST10_GlobalError".SafetyDoor.MaterialDoor.NotLock_2 OR "ST10_GlobalError".SafetyDoor.MaterialDoor.NotLock_1) AND "Station_Sys".Auto.Running THEN
       "AutoProcessControl".Status.HShaftLifting.Status := 2;
   END_IF;
   IF "AlwaysTRUE" AND "Station_Sys".Interface.Reset THEN
       "AutoProcessControl".Status.HShaftLifting.Status := 0;
   END_IF;
END_REGION

REGION Network 50: loading Stop 1 timeout
   RUNG wire#powerrail
      Contact( "AlwaysTRUE" )
      Contact( "ST10_Flow25_HShaftLoad&Unload_iDB".WaitPalletArrveNextPos.X )
      I_Contact( "iH-shaftLoadingDetection2" )
      { S7_Templates := "time_type := Time" } "TON".TON[2].TON(pt := t#8s, et =>)
      S_Coil( "ST10_DeviceError".H.ShaftLine.LoadingStop1timeout )
   END_RUNG
   // the same network as SCL:
   "TON".TON[2].TON(IN := "AlwaysTRUE" AND "ST10_Flow25_HShaftLoad&Unload_iDB".WaitPalletArrveNextPos.X AND NOT "iH-shaftLoadingDetection2",
                    PT := t#8s);
   IF "TON".TON[2].Q THEN "ST10_DeviceError".H.ShaftLine.LoadingStop1timeout := TRUE; END_IF;
END_REGION

REGION Network 51: loading Stop 2 timeout
   RUNG wire#powerrail
      Contact( "AlwaysTRUE" )
      Contact( "ST10_Flow25_HShaftLoad&Unload_iDB".WaitPalletArrveNextPos_1.X )
      I_Contact( "iH-shaftLoadingDetection3" )
      { S7_Templates := "time_type := Time" } "TON".TON[3].TON(pt := t#8s, et =>)
      S_Coil( "ST10_DeviceError".H.ShaftLine.LoadingStop2timeout )
   END_RUNG
   // the same network as SCL:
   "TON".TON[3].TON(IN := "AlwaysTRUE" AND "ST10_Flow25_HShaftLoad&Unload_iDB".WaitPalletArrveNextPos_1.X AND NOT "iH-shaftLoadingDetection3",
                    PT := t#8s);
   IF "TON".TON[3].Q THEN "ST10_DeviceError".H.ShaftLine.LoadingStop2timeout := TRUE; END_IF;
END_REGION

REGION Network 52: loading Stop 3 timeout
   RUNG wire#powerrail
      Contact( "AlwaysTRUE" )
      Contact( "ST10_Flow25_HShaftLoad&Unload_iDB".WaitPalletArrveNextPos_2.X )
      I_Contact( "iH-shaftLoadingDetection4" )
      { S7_Templates := "time_type := Time" } "TON".TON[4].TON(pt := t#8s, et =>)
      S_Coil( "ST10_DeviceError".H.ShaftLine.LoadingStop3timeout )
   END_RUNG
   // the same network as SCL:
   "TON".TON[4].TON(IN := "AlwaysTRUE" AND "ST10_Flow25_HShaftLoad&Unload_iDB".WaitPalletArrveNextPos_2.X AND NOT "iH-shaftLoadingDetection4",
                    PT := t#8s);
   IF "TON".TON[4].Q THEN "ST10_DeviceError".H.ShaftLine.LoadingStop3timeout := TRUE; END_IF;
END_REGION

REGION Network 53: loading Stop 4 timeout
   RUNG wire#powerrail
      Contact( "AlwaysTRUE" )
      Contact( "ST10_Flow25_HShaftLoad&Unload_iDB".WaitPalletArrveNextPos_3.X )
      I_Contact( "iH-shaftLiftingPalletDischarge" )
      { S7_Templates := "time_type := Time" } "TON".TON[9].TON(pt := t#8s, et =>)
      S_Coil( "ST10_DeviceError".H.ShaftLine.LoadingStop4timeout )
   END_RUNG
   // the same network as SCL:
   "TON".TON[9].TON(IN := "AlwaysTRUE" AND "ST10_Flow25_HShaftLoad&Unload_iDB".WaitPalletArrveNextPos_3.X AND NOT "iH-shaftLiftingPalletDischarge",
                    PT := t#8s);
   IF "TON".TON[9].Q THEN "ST10_DeviceError".H.ShaftLine.LoadingStop4timeout := TRUE; END_IF;
END_REGION

REGION Network 54: unLoading Stop1 timeout
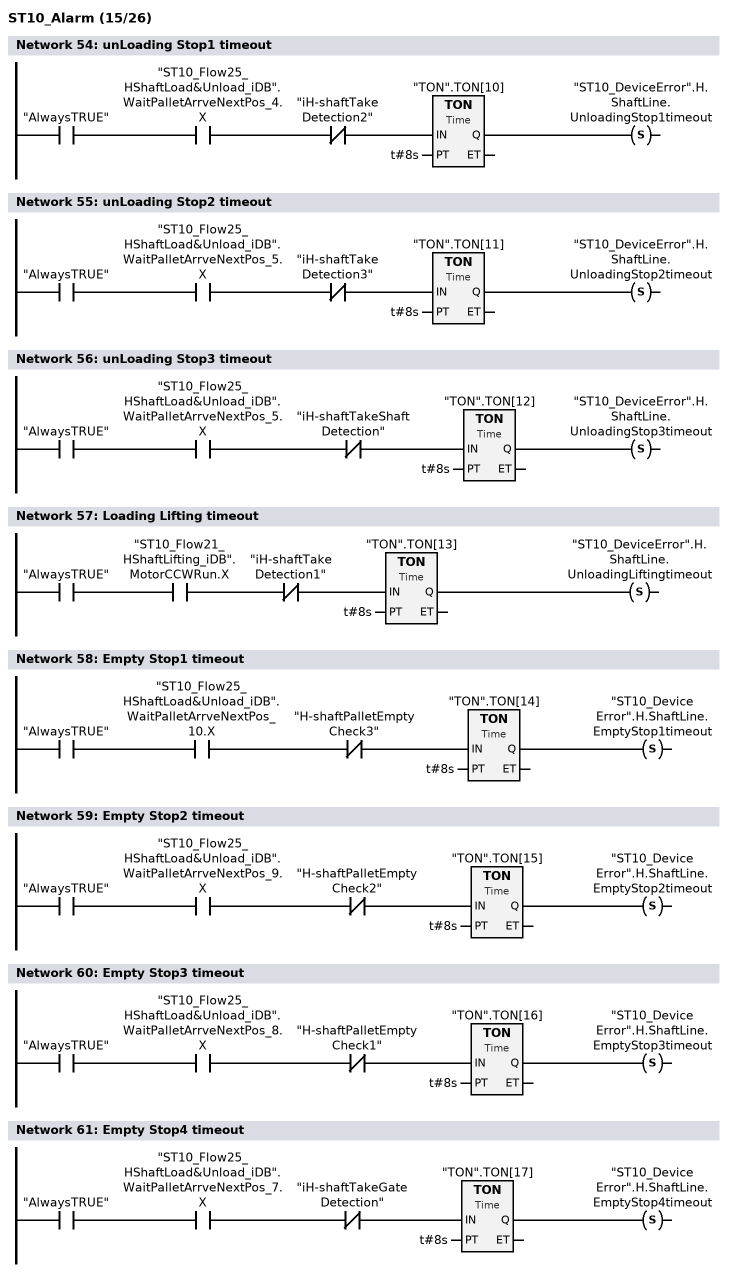
   RUNG wire#powerrail
      Contact( "AlwaysTRUE" )
      Contact( "ST10_Flow25_HShaftLoad&Unload_iDB".WaitPalletArrveNextPos_4.X )
      I_Contact( "iH-shaftTakeDetection2" )
      { S7_Templates := "time_type := Time" } "TON".TON[10].TON(pt := t#8s, et =>)
      S_Coil( "ST10_DeviceError".H.ShaftLine.UnloadingStop1timeout )
   END_RUNG
   // the same network as SCL:
   "TON".TON[10].TON(IN := "AlwaysTRUE" AND "ST10_Flow25_HShaftLoad&Unload_iDB".WaitPalletArrveNextPos_4.X AND NOT "iH-shaftTakeDetection2",
                     PT := t#8s);
   IF "TON".TON[10].Q THEN "ST10_DeviceError".H.ShaftLine.UnloadingStop1timeout := TRUE; END_IF;
END_REGION

REGION Network 55: unLoading Stop2 timeout
   RUNG wire#powerrail
      Contact( "AlwaysTRUE" )
      Contact( "ST10_Flow25_HShaftLoad&Unload_iDB".WaitPalletArrveNextPos_5.X )
      I_Contact( "iH-shaftTakeDetection3" )
      { S7_Templates := "time_type := Time" } "TON".TON[11].TON(pt := t#8s, et =>)
      S_Coil( "ST10_DeviceError".H.ShaftLine.UnloadingStop2timeout )
   END_RUNG
   // the same network as SCL:
   "TON".TON[11].TON(IN := "AlwaysTRUE" AND "ST10_Flow25_HShaftLoad&Unload_iDB".WaitPalletArrveNextPos_5.X AND NOT "iH-shaftTakeDetection3",
                     PT := t#8s);
   IF "TON".TON[11].Q THEN "ST10_DeviceError".H.ShaftLine.UnloadingStop2timeout := TRUE; END_IF;
END_REGION

REGION Network 56: unLoading Stop3 timeout
   RUNG wire#powerrail
      Contact( "AlwaysTRUE" )
      Contact( "ST10_Flow25_HShaftLoad&Unload_iDB".WaitPalletArrveNextPos_5.X )
      I_Contact( "iH-shaftTakeShaftDetection" )
      { S7_Templates := "time_type := Time" } "TON".TON[12].TON(pt := t#8s, et =>)
      S_Coil( "ST10_DeviceError".H.ShaftLine.UnloadingStop3timeout )
   END_RUNG
   // the same network as SCL:
   "TON".TON[12].TON(IN := "AlwaysTRUE" AND "ST10_Flow25_HShaftLoad&Unload_iDB".WaitPalletArrveNextPos_5.X AND NOT "iH-shaftTakeShaftDetection",
                     PT := t#8s);
   IF "TON".TON[12].Q THEN "ST10_DeviceError".H.ShaftLine.UnloadingStop3timeout := TRUE; END_IF;
END_REGION

REGION Network 57: Loading Lifting timeout
   RUNG wire#powerrail
      Contact( "AlwaysTRUE" )
      Contact( "ST10_Flow21_HShaftLifting_iDB".MotorCCWRun.X )
      I_Contact( "iH-shaftTakeDetection1" )
      { S7_Templates := "time_type := Time" } "TON".TON[13].TON(pt := t#8s, et =>)
      S_Coil( "ST10_DeviceError".H.ShaftLine.UnloadingLiftingtimeout )
   END_RUNG
   // the same network as SCL:
   "TON".TON[13].TON(IN := "AlwaysTRUE" AND "ST10_Flow21_HShaftLifting_iDB".MotorCCWRun.X AND NOT "iH-shaftTakeDetection1",
                     PT := t#8s);
   IF "TON".TON[13].Q THEN "ST10_DeviceError".H.ShaftLine.UnloadingLiftingtimeout := TRUE; END_IF;
END_REGION

REGION Network 58: Empty Stop1 timeout
   RUNG wire#powerrail
      Contact( "AlwaysTRUE" )
      Contact( "ST10_Flow25_HShaftLoad&Unload_iDB".WaitPalletArrveNextPos_10.X )
      I_Contact( "H-shaftPalletEmptyCheck3" )
      { S7_Templates := "time_type := Time" } "TON".TON[14].TON(pt := t#8s, et =>)
      S_Coil( "ST10_DeviceError".H.ShaftLine.EmptyStop1timeout )
   END_RUNG
   // the same network as SCL:
   "TON".TON[14].TON(IN := "AlwaysTRUE" AND "ST10_Flow25_HShaftLoad&Unload_iDB".WaitPalletArrveNextPos_10.X AND NOT "H-shaftPalletEmptyCheck3",
                     PT := t#8s);
   IF "TON".TON[14].Q THEN "ST10_DeviceError".H.ShaftLine.EmptyStop1timeout := TRUE; END_IF;
END_REGION

REGION Network 59: Empty Stop2 timeout
   RUNG wire#powerrail
      Contact( "AlwaysTRUE" )
      Contact( "ST10_Flow25_HShaftLoad&Unload_iDB".WaitPalletArrveNextPos_9.X )
      I_Contact( "H-shaftPalletEmptyCheck2" )
      { S7_Templates := "time_type := Time" } "TON".TON[15].TON(pt := t#8s, et =>)
      S_Coil( "ST10_DeviceError".H.ShaftLine.EmptyStop2timeout )
   END_RUNG
   // the same network as SCL:
   "TON".TON[15].TON(IN := "AlwaysTRUE" AND "ST10_Flow25_HShaftLoad&Unload_iDB".WaitPalletArrveNextPos_9.X AND NOT "H-shaftPalletEmptyCheck2",
                     PT := t#8s);
   IF "TON".TON[15].Q THEN "ST10_DeviceError".H.ShaftLine.EmptyStop2timeout := TRUE; END_IF;
END_REGION

REGION Network 60: Empty Stop3 timeout
   RUNG wire#powerrail
      Contact( "AlwaysTRUE" )
      Contact( "ST10_Flow25_HShaftLoad&Unload_iDB".WaitPalletArrveNextPos_8.X )
      I_Contact( "H-shaftPalletEmptyCheck1" )
      { S7_Templates := "time_type := Time" } "TON".TON[16].TON(pt := t#8s, et =>)
      S_Coil( "ST10_DeviceError".H.ShaftLine.EmptyStop3timeout )
   END_RUNG
   // the same network as SCL:
   "TON".TON[16].TON(IN := "AlwaysTRUE" AND "ST10_Flow25_HShaftLoad&Unload_iDB".WaitPalletArrveNextPos_8.X AND NOT "H-shaftPalletEmptyCheck1",
                     PT := t#8s);
   IF "TON".TON[16].Q THEN "ST10_DeviceError".H.ShaftLine.EmptyStop3timeout := TRUE; END_IF;
END_REGION

REGION Network 61: Empty Stop4 timeout
   RUNG wire#powerrail
      Contact( "AlwaysTRUE" )
      Contact( "ST10_Flow25_HShaftLoad&Unload_iDB".WaitPalletArrveNextPos_7.X )
      I_Contact( "iH-shaftTakeGateDetection" )
      { S7_Templates := "time_type := Time" } "TON".TON[17].TON(pt := t#8s, et =>)
      S_Coil( "ST10_DeviceError".H.ShaftLine.EmptyStop4timeout )
   END_RUNG
   // the same network as SCL:
   "TON".TON[17].TON(IN := "AlwaysTRUE" AND "ST10_Flow25_HShaftLoad&Unload_iDB".WaitPalletArrveNextPos_7.X AND NOT "iH-shaftTakeGateDetection",
                     PT := t#8s);
   IF "TON".TON[17].Q THEN "ST10_DeviceError".H.ShaftLine.EmptyStop4timeout := TRUE; END_IF;
END_REGION

REGION Network 63: ******************** J_Magnet loading ********************
END_REGION

REGION Network 64: J
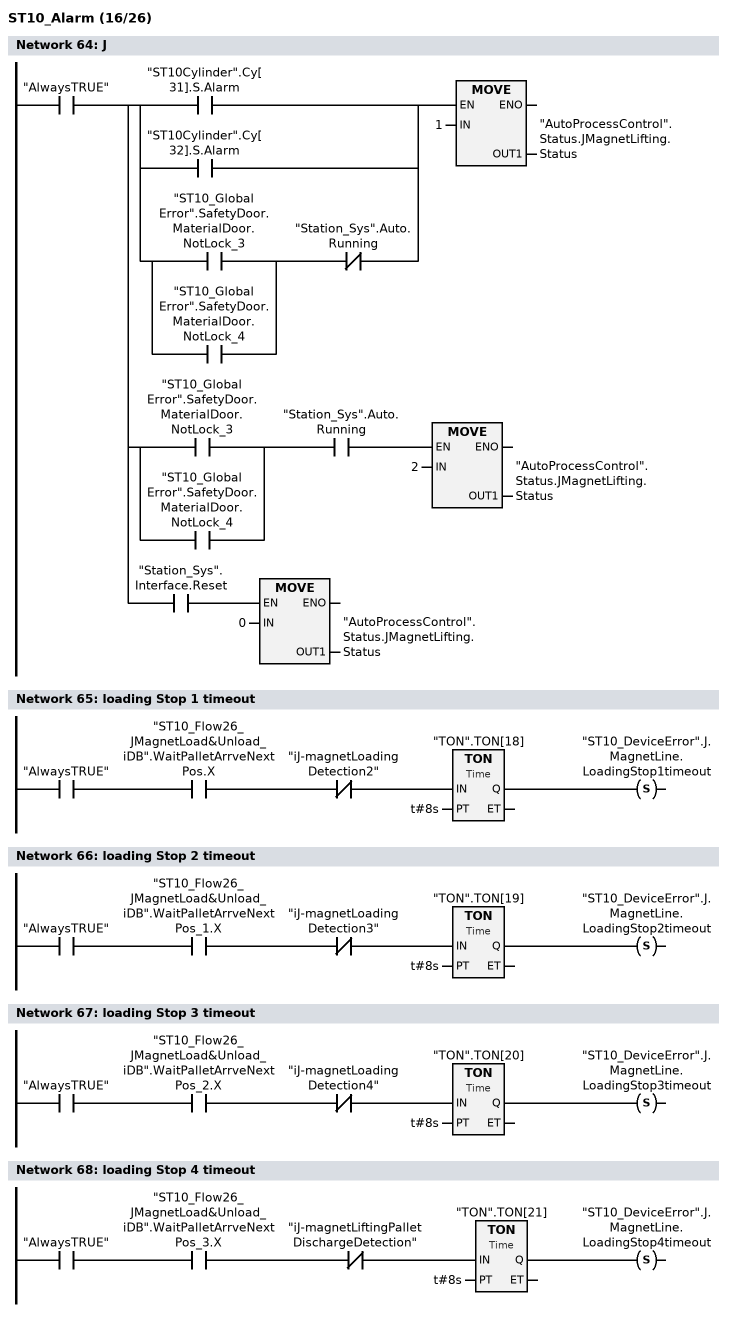
   RUNG wire#powerrail
      Contact( "AlwaysTRUE" )
      wire#w1
      Contact( "ST10Cylinder".Cy[31].S.Alarm )
      wire#w2
      Move(in := 1, out1 => "AutoProcessControl".Status.JMagnetLifting.Status)
   END_RUNG
   RUNG wire#w1
      Contact( "ST10Cylinder".Cy[32].S.Alarm )
   END_RUNG wire#w2
   RUNG wire#w1
      Contact( "ST10_GlobalError".SafetyDoor.MaterialDoor.NotLock_3 )
      wire#w3
      I_Contact( "Station_Sys".Auto.Running )
   END_RUNG wire#w2
   RUNG wire#w1
      Contact( "ST10_GlobalError".SafetyDoor.MaterialDoor.NotLock_4 )
   END_RUNG wire#w3
   RUNG wire#w1
      Contact( "ST10_GlobalError".SafetyDoor.MaterialDoor.NotLock_3 )
      wire#w4
      Contact( "Station_Sys".Auto.Running )
      Move(in := 2, out1 => "AutoProcessControl".Status.JMagnetLifting.Status)
   END_RUNG
   RUNG wire#w1
      Contact( "ST10_GlobalError".SafetyDoor.MaterialDoor.NotLock_4 )
   END_RUNG wire#w4
   RUNG wire#w1
      Contact( "Station_Sys".Interface.Reset )
      Move(in := 0, out1 => "AutoProcessControl".Status.JMagnetLifting.Status)
   END_RUNG
   // the same network as SCL:
   IF "AlwaysTRUE" AND ("ST10Cylinder".Cy[31].S.Alarm OR "ST10Cylinder".Cy[32].S.Alarm OR (("ST10_GlobalError".SafetyDoor.MaterialDoor.NotLock_3 OR "ST10_GlobalError".SafetyDoor.MaterialDoor.NotLock_4) AND NOT "Station_Sys".Auto.Running)) THEN
       "AutoProcessControl".Status.JMagnetLifting.Status := 1;
   END_IF;
   IF "AlwaysTRUE" AND ("ST10_GlobalError".SafetyDoor.MaterialDoor.NotLock_3 OR "ST10_GlobalError".SafetyDoor.MaterialDoor.NotLock_4) AND "Station_Sys".Auto.Running THEN
       "AutoProcessControl".Status.JMagnetLifting.Status := 2;
   END_IF;
   IF "AlwaysTRUE" AND "Station_Sys".Interface.Reset THEN
       "AutoProcessControl".Status.JMagnetLifting.Status := 0;
   END_IF;
END_REGION

REGION Network 65: loading Stop 1 timeout
   RUNG wire#powerrail
      Contact( "AlwaysTRUE" )
      Contact( "ST10_Flow26_JMagnetLoad&Unload_iDB".WaitPalletArrveNextPos.X )
      I_Contact( "iJ-magnetLoadingDetection2" )
      { S7_Templates := "time_type := Time" } "TON".TON[18].TON(pt := t#8s, et =>)
      S_Coil( "ST10_DeviceError".J.MagnetLine.LoadingStop1timeout )
   END_RUNG
   // the same network as SCL:
   "TON".TON[18].TON(IN := "AlwaysTRUE" AND "ST10_Flow26_JMagnetLoad&Unload_iDB".WaitPalletArrveNextPos.X AND NOT "iJ-magnetLoadingDetection2",
                     PT := t#8s);
   IF "TON".TON[18].Q THEN "ST10_DeviceError".J.MagnetLine.LoadingStop1timeout := TRUE; END_IF;
END_REGION

REGION Network 66: loading Stop 2 timeout
   RUNG wire#powerrail
      Contact( "AlwaysTRUE" )
      Contact( "ST10_Flow26_JMagnetLoad&Unload_iDB".WaitPalletArrveNextPos_1.X )
      I_Contact( "iJ-magnetLoadingDetection3" )
      { S7_Templates := "time_type := Time" } "TON".TON[19].TON(pt := t#8s, et =>)
      S_Coil( "ST10_DeviceError".J.MagnetLine.LoadingStop2timeout )
   END_RUNG
   // the same network as SCL:
   "TON".TON[19].TON(IN := "AlwaysTRUE" AND "ST10_Flow26_JMagnetLoad&Unload_iDB".WaitPalletArrveNextPos_1.X AND NOT "iJ-magnetLoadingDetection3",
                     PT := t#8s);
   IF "TON".TON[19].Q THEN "ST10_DeviceError".J.MagnetLine.LoadingStop2timeout := TRUE; END_IF;
END_REGION

REGION Network 67: loading Stop 3 timeout
   RUNG wire#powerrail
      Contact( "AlwaysTRUE" )
      Contact( "ST10_Flow26_JMagnetLoad&Unload_iDB".WaitPalletArrveNextPos_2.X )
      I_Contact( "iJ-magnetLoadingDetection4" )
      { S7_Templates := "time_type := Time" } "TON".TON[20].TON(pt := t#8s, et =>)
      S_Coil( "ST10_DeviceError".J.MagnetLine.LoadingStop3timeout )
   END_RUNG
   // the same network as SCL:
   "TON".TON[20].TON(IN := "AlwaysTRUE" AND "ST10_Flow26_JMagnetLoad&Unload_iDB".WaitPalletArrveNextPos_2.X AND NOT "iJ-magnetLoadingDetection4",
                     PT := t#8s);
   IF "TON".TON[20].Q THEN "ST10_DeviceError".J.MagnetLine.LoadingStop3timeout := TRUE; END_IF;
END_REGION

REGION Network 68: loading Stop 4 timeout
   RUNG wire#powerrail
      Contact( "AlwaysTRUE" )
      Contact( "ST10_Flow26_JMagnetLoad&Unload_iDB".WaitPalletArrveNextPos_3.X )
      I_Contact( "iJ-magnetLiftingPalletDischargeDetection" )
      { S7_Templates := "time_type := Time" } "TON".TON[21].TON(pt := t#8s, et =>)
      S_Coil( "ST10_DeviceError".J.MagnetLine.LoadingStop4timeout )
   END_RUNG
   // the same network as SCL:
   "TON".TON[21].TON(IN := "AlwaysTRUE" AND "ST10_Flow26_JMagnetLoad&Unload_iDB".WaitPalletArrveNextPos_3.X AND NOT "iJ-magnetLiftingPalletDischargeDetection",
                     PT := t#8s);
   IF "TON".TON[21].Q THEN "ST10_DeviceError".J.MagnetLine.LoadingStop4timeout := TRUE; END_IF;
END_REGION

REGION Network 69: unLoading Stop1 timeout
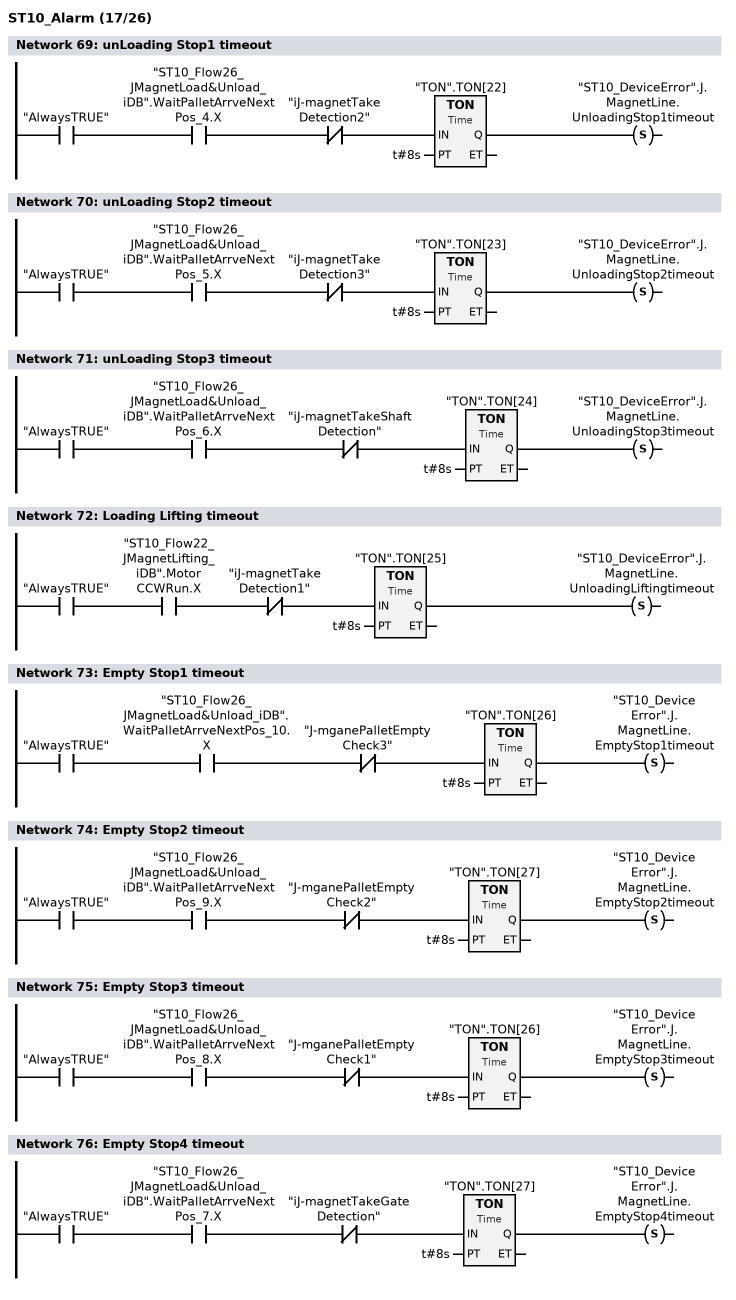
   RUNG wire#powerrail
      Contact( "AlwaysTRUE" )
      Contact( "ST10_Flow26_JMagnetLoad&Unload_iDB".WaitPalletArrveNextPos_4.X )
      I_Contact( "iJ-magnetTakeDetection2" )
      { S7_Templates := "time_type := Time" } "TON".TON[22].TON(pt := t#8s, et =>)
      S_Coil( "ST10_DeviceError".J.MagnetLine.UnloadingStop1timeout )
   END_RUNG
   // the same network as SCL:
   "TON".TON[22].TON(IN := "AlwaysTRUE" AND "ST10_Flow26_JMagnetLoad&Unload_iDB".WaitPalletArrveNextPos_4.X AND NOT "iJ-magnetTakeDetection2",
                     PT := t#8s);
   IF "TON".TON[22].Q THEN "ST10_DeviceError".J.MagnetLine.UnloadingStop1timeout := TRUE; END_IF;
END_REGION

REGION Network 70: unLoading Stop2 timeout
   RUNG wire#powerrail
      Contact( "AlwaysTRUE" )
      Contact( "ST10_Flow26_JMagnetLoad&Unload_iDB".WaitPalletArrveNextPos_5.X )
      I_Contact( "iJ-magnetTakeDetection3" )
      { S7_Templates := "time_type := Time" } "TON".TON[23].TON(pt := t#8s, et =>)
      S_Coil( "ST10_DeviceError".J.MagnetLine.UnloadingStop2timeout )
   END_RUNG
   // the same network as SCL:
   "TON".TON[23].TON(IN := "AlwaysTRUE" AND "ST10_Flow26_JMagnetLoad&Unload_iDB".WaitPalletArrveNextPos_5.X AND NOT "iJ-magnetTakeDetection3",
                     PT := t#8s);
   IF "TON".TON[23].Q THEN "ST10_DeviceError".J.MagnetLine.UnloadingStop2timeout := TRUE; END_IF;
END_REGION

REGION Network 71: unLoading Stop3 timeout
   RUNG wire#powerrail
      Contact( "AlwaysTRUE" )
      Contact( "ST10_Flow26_JMagnetLoad&Unload_iDB".WaitPalletArrveNextPos_6.X )
      I_Contact( "iJ-magnetTakeShaftDetection" )
      { S7_Templates := "time_type := Time" } "TON".TON[24].TON(pt := t#8s, et =>)
      S_Coil( "ST10_DeviceError".J.MagnetLine.UnloadingStop3timeout )
   END_RUNG
   // the same network as SCL:
   "TON".TON[24].TON(IN := "AlwaysTRUE" AND "ST10_Flow26_JMagnetLoad&Unload_iDB".WaitPalletArrveNextPos_6.X AND NOT "iJ-magnetTakeShaftDetection",
                     PT := t#8s);
   IF "TON".TON[24].Q THEN "ST10_DeviceError".J.MagnetLine.UnloadingStop3timeout := TRUE; END_IF;
END_REGION

REGION Network 72: Loading Lifting timeout
   RUNG wire#powerrail
      Contact( "AlwaysTRUE" )
      Contact( "ST10_Flow22_JMagnetLifting_iDB".MotorCCWRun.X )
      I_Contact( "iJ-magnetTakeDetection1" )
      { S7_Templates := "time_type := Time" } "TON".TON[25].TON(pt := t#8s, et =>)
      S_Coil( "ST10_DeviceError".J.MagnetLine.UnloadingLiftingtimeout )
   END_RUNG
   // the same network as SCL:
   "TON".TON[25].TON(IN := "AlwaysTRUE" AND "ST10_Flow22_JMagnetLifting_iDB".MotorCCWRun.X AND NOT "iJ-magnetTakeDetection1",
                     PT := t#8s);
   IF "TON".TON[25].Q THEN "ST10_DeviceError".J.MagnetLine.UnloadingLiftingtimeout := TRUE; END_IF;
END_REGION

REGION Network 73: Empty Stop1 timeout
   RUNG wire#powerrail
      Contact( "AlwaysTRUE" )
      Contact( "ST10_Flow26_JMagnetLoad&Unload_iDB".WaitPalletArrveNextPos_10.X )
      I_Contact( "J-mganePalletEmptyCheck3" )
      { S7_Templates := "time_type := Time" } "TON".TON[26].TON(pt := t#8s, et =>)
      S_Coil( "ST10_DeviceError".J.MagnetLine.EmptyStop1timeout )
   END_RUNG
   // the same network as SCL:
   "TON".TON[26].TON(IN := "AlwaysTRUE" AND "ST10_Flow26_JMagnetLoad&Unload_iDB".WaitPalletArrveNextPos_10.X AND NOT "J-mganePalletEmptyCheck3",
                     PT := t#8s);
   IF "TON".TON[26].Q THEN "ST10_DeviceError".J.MagnetLine.EmptyStop1timeout := TRUE; END_IF;
END_REGION

REGION Network 74: Empty Stop2 timeout
   RUNG wire#powerrail
      Contact( "AlwaysTRUE" )
      Contact( "ST10_Flow26_JMagnetLoad&Unload_iDB".WaitPalletArrveNextPos_9.X )
      I_Contact( "J-mganePalletEmptyCheck2" )
      { S7_Templates := "time_type := Time" } "TON".TON[27].TON(pt := t#8s, et =>)
      S_Coil( "ST10_DeviceError".J.MagnetLine.EmptyStop2timeout )
   END_RUNG
   // the same network as SCL:
   "TON".TON[27].TON(IN := "AlwaysTRUE" AND "ST10_Flow26_JMagnetLoad&Unload_iDB".WaitPalletArrveNextPos_9.X AND NOT "J-mganePalletEmptyCheck2",
                     PT := t#8s);
   IF "TON".TON[27].Q THEN "ST10_DeviceError".J.MagnetLine.EmptyStop2timeout := TRUE; END_IF;
END_REGION

REGION Network 75: Empty Stop3 timeout
   RUNG wire#powerrail
      Contact( "AlwaysTRUE" )
      Contact( "ST10_Flow26_JMagnetLoad&Unload_iDB".WaitPalletArrveNextPos_8.X )
      I_Contact( "J-mganePalletEmptyCheck1" )
      { S7_Templates := "time_type := Time" } "TON".TON[26].TON(pt := t#8s, et =>)
      S_Coil( "ST10_DeviceError".J.MagnetLine.EmptyStop3timeout )
   END_RUNG
   // the same network as SCL:
   "TON".TON[26].TON(IN := "AlwaysTRUE" AND "ST10_Flow26_JMagnetLoad&Unload_iDB".WaitPalletArrveNextPos_8.X AND NOT "J-mganePalletEmptyCheck1",
                     PT := t#8s);
   IF "TON".TON[26].Q THEN "ST10_DeviceError".J.MagnetLine.EmptyStop3timeout := TRUE; END_IF;
END_REGION

REGION Network 76: Empty Stop4 timeout
   RUNG wire#powerrail
      Contact( "AlwaysTRUE" )
      Contact( "ST10_Flow26_JMagnetLoad&Unload_iDB".WaitPalletArrveNextPos_7.X )
      I_Contact( "iJ-magnetTakeGateDetection" )
      { S7_Templates := "time_type := Time" } "TON".TON[27].TON(pt := t#8s, et =>)
      S_Coil( "ST10_DeviceError".J.MagnetLine.EmptyStop4timeout )
   END_RUNG
   // the same network as SCL:
   "TON".TON[27].TON(IN := "AlwaysTRUE" AND "ST10_Flow26_JMagnetLoad&Unload_iDB".WaitPalletArrveNextPos_7.X AND NOT "iJ-magnetTakeGateDetection",
                     PT := t#8s);
   IF "TON".TON[27].Q THEN "ST10_DeviceError".J.MagnetLine.EmptyStop4timeout := TRUE; END_IF;
END_REGION

REGION Network 78: ******************** K_Reserve loading ********************
END_REGION

REGION Network 79: K
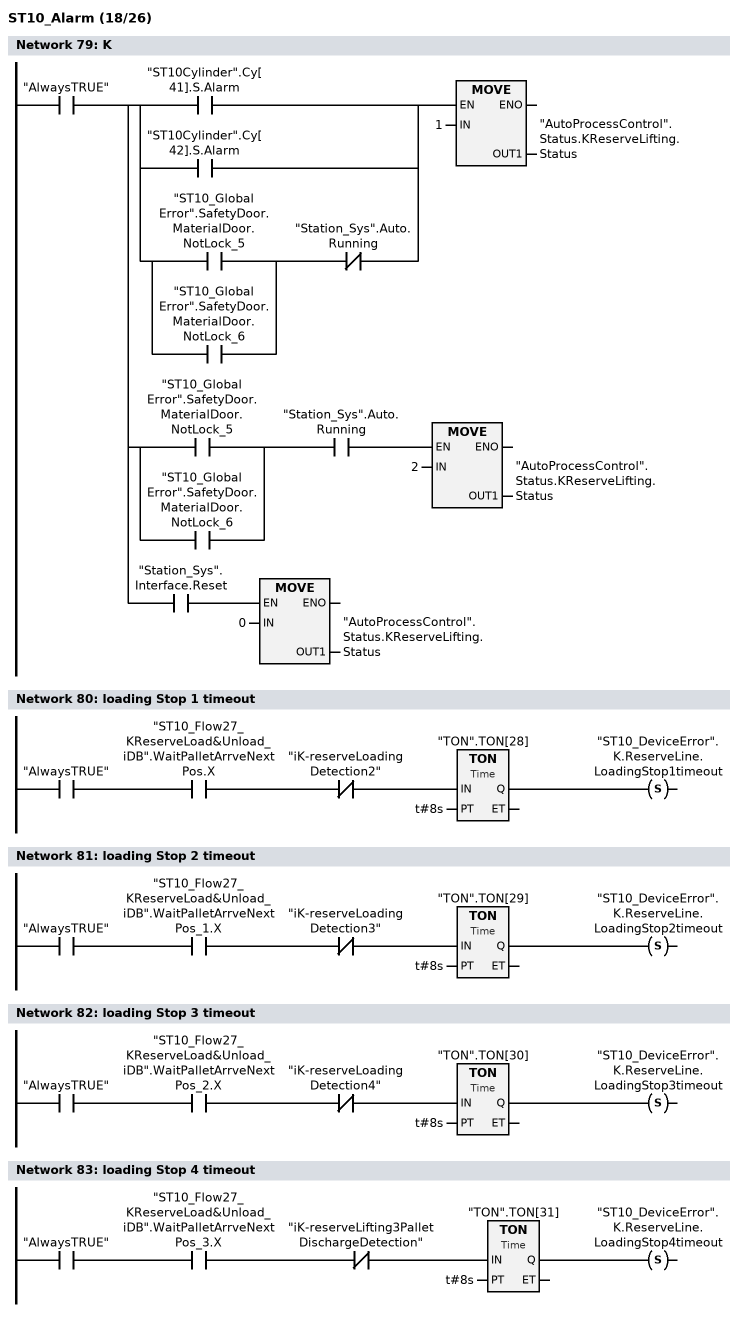
   RUNG wire#powerrail
      Contact( "AlwaysTRUE" )
      wire#w1
      Contact( "ST10Cylinder".Cy[41].S.Alarm )
      wire#w2
      Move(in := 1, out1 => "AutoProcessControl".Status.KReserveLifting.Status)
   END_RUNG
   RUNG wire#w1
      Contact( "ST10Cylinder".Cy[42].S.Alarm )
   END_RUNG wire#w2
   RUNG wire#w1
      Contact( "ST10_GlobalError".SafetyDoor.MaterialDoor.NotLock_5 )
      wire#w3
      I_Contact( "Station_Sys".Auto.Running )
   END_RUNG wire#w2
   RUNG wire#w1
      Contact( "ST10_GlobalError".SafetyDoor.MaterialDoor.NotLock_6 )
   END_RUNG wire#w3
   RUNG wire#w1
      Contact( "ST10_GlobalError".SafetyDoor.MaterialDoor.NotLock_5 )
      wire#w4
      Contact( "Station_Sys".Auto.Running )
      Move(in := 2, out1 => "AutoProcessControl".Status.KReserveLifting.Status)
   END_RUNG
   RUNG wire#w1
      Contact( "ST10_GlobalError".SafetyDoor.MaterialDoor.NotLock_6 )
   END_RUNG wire#w4
   RUNG wire#w1
      Contact( "Station_Sys".Interface.Reset )
      Move(in := 0, out1 => "AutoProcessControl".Status.KReserveLifting.Status)
   END_RUNG
   // the same network as SCL:
   IF "AlwaysTRUE" AND ("ST10Cylinder".Cy[41].S.Alarm OR "ST10Cylinder".Cy[42].S.Alarm OR (("ST10_GlobalError".SafetyDoor.MaterialDoor.NotLock_5 OR "ST10_GlobalError".SafetyDoor.MaterialDoor.NotLock_6) AND NOT "Station_Sys".Auto.Running)) THEN
       "AutoProcessControl".Status.KReserveLifting.Status := 1;
   END_IF;
   IF "AlwaysTRUE" AND ("ST10_GlobalError".SafetyDoor.MaterialDoor.NotLock_5 OR "ST10_GlobalError".SafetyDoor.MaterialDoor.NotLock_6) AND "Station_Sys".Auto.Running THEN
       "AutoProcessControl".Status.KReserveLifting.Status := 2;
   END_IF;
   IF "AlwaysTRUE" AND "Station_Sys".Interface.Reset THEN
       "AutoProcessControl".Status.KReserveLifting.Status := 0;
   END_IF;
END_REGION

REGION Network 80: loading Stop 1 timeout
   RUNG wire#powerrail
      Contact( "AlwaysTRUE" )
      Contact( "ST10_Flow27_KReserveLoad&Unload_iDB".WaitPalletArrveNextPos.X )
      I_Contact( "iK-reserveLoadingDetection2" )
      { S7_Templates := "time_type := Time" } "TON".TON[28].TON(pt := t#8s, et =>)
      S_Coil( "ST10_DeviceError".K.ReserveLine.LoadingStop1timeout )
   END_RUNG
   // the same network as SCL:
   "TON".TON[28].TON(IN := "AlwaysTRUE" AND "ST10_Flow27_KReserveLoad&Unload_iDB".WaitPalletArrveNextPos.X AND NOT "iK-reserveLoadingDetection2",
                     PT := t#8s);
   IF "TON".TON[28].Q THEN "ST10_DeviceError".K.ReserveLine.LoadingStop1timeout := TRUE; END_IF;
END_REGION

REGION Network 81: loading Stop 2 timeout
   RUNG wire#powerrail
      Contact( "AlwaysTRUE" )
      Contact( "ST10_Flow27_KReserveLoad&Unload_iDB".WaitPalletArrveNextPos_1.X )
      I_Contact( "iK-reserveLoadingDetection3" )
      { S7_Templates := "time_type := Time" } "TON".TON[29].TON(pt := t#8s, et =>)
      S_Coil( "ST10_DeviceError".K.ReserveLine.LoadingStop2timeout )
   END_RUNG
   // the same network as SCL:
   "TON".TON[29].TON(IN := "AlwaysTRUE" AND "ST10_Flow27_KReserveLoad&Unload_iDB".WaitPalletArrveNextPos_1.X AND NOT "iK-reserveLoadingDetection3",
                     PT := t#8s);
   IF "TON".TON[29].Q THEN "ST10_DeviceError".K.ReserveLine.LoadingStop2timeout := TRUE; END_IF;
END_REGION

REGION Network 82: loading Stop 3 timeout
   RUNG wire#powerrail
      Contact( "AlwaysTRUE" )
      Contact( "ST10_Flow27_KReserveLoad&Unload_iDB".WaitPalletArrveNextPos_2.X )
      I_Contact( "iK-reserveLoadingDetection4" )
      { S7_Templates := "time_type := Time" } "TON".TON[30].TON(pt := t#8s, et =>)
      S_Coil( "ST10_DeviceError".K.ReserveLine.LoadingStop3timeout )
   END_RUNG
   // the same network as SCL:
   "TON".TON[30].TON(IN := "AlwaysTRUE" AND "ST10_Flow27_KReserveLoad&Unload_iDB".WaitPalletArrveNextPos_2.X AND NOT "iK-reserveLoadingDetection4",
                     PT := t#8s);
   IF "TON".TON[30].Q THEN "ST10_DeviceError".K.ReserveLine.LoadingStop3timeout := TRUE; END_IF;
END_REGION

REGION Network 83: loading Stop 4 timeout
   RUNG wire#powerrail
      Contact( "AlwaysTRUE" )
      Contact( "ST10_Flow27_KReserveLoad&Unload_iDB".WaitPalletArrveNextPos_3.X )
      I_Contact( "iK-reserveLifting3PalletDischargeDetection" )
      { S7_Templates := "time_type := Time" } "TON".TON[31].TON(pt := t#8s, et =>)
      S_Coil( "ST10_DeviceError".K.ReserveLine.LoadingStop4timeout )
   END_RUNG
   // the same network as SCL:
   "TON".TON[31].TON(IN := "AlwaysTRUE" AND "ST10_Flow27_KReserveLoad&Unload_iDB".WaitPalletArrveNextPos_3.X AND NOT "iK-reserveLifting3PalletDischargeDetection",
                     PT := t#8s);
   IF "TON".TON[31].Q THEN "ST10_DeviceError".K.ReserveLine.LoadingStop4timeout := TRUE; END_IF;
END_REGION

REGION Network 84: unLoading Stop1 timeout
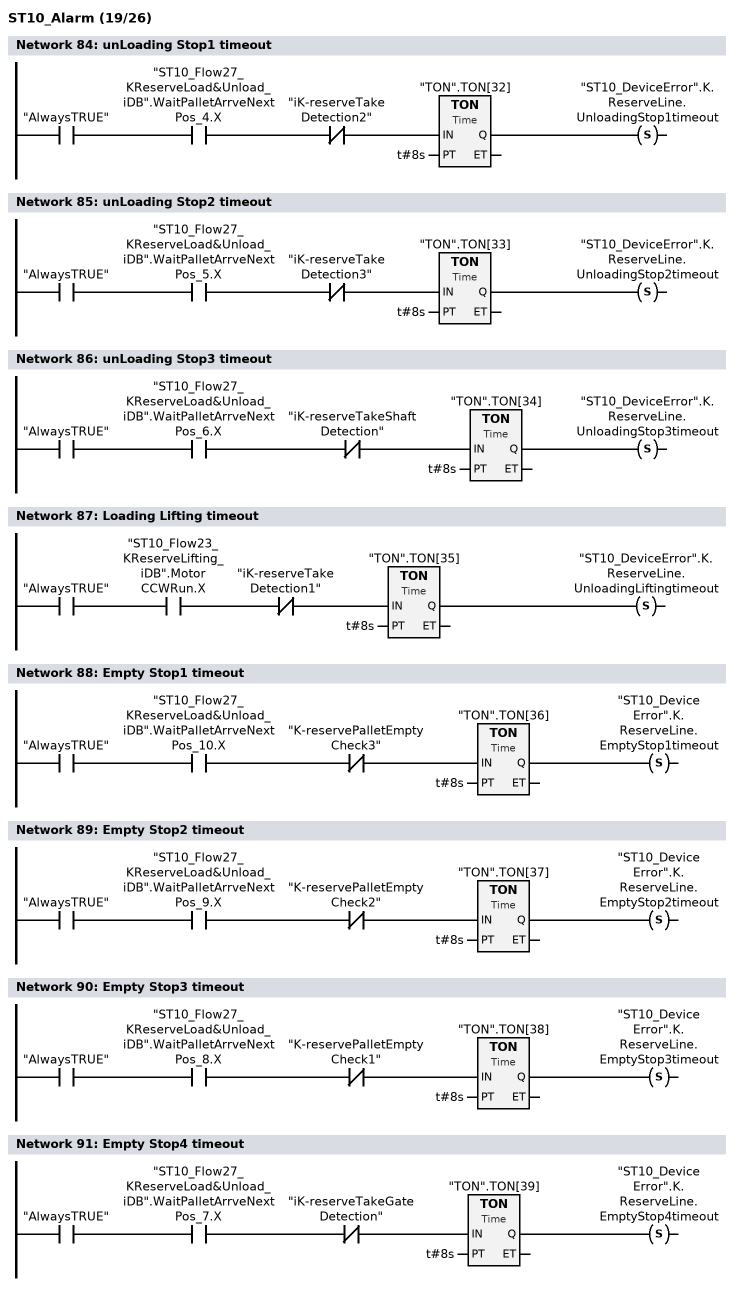
   RUNG wire#powerrail
      Contact( "AlwaysTRUE" )
      Contact( "ST10_Flow27_KReserveLoad&Unload_iDB".WaitPalletArrveNextPos_4.X )
      I_Contact( "iK-reserveTakeDetection2" )
      { S7_Templates := "time_type := Time" } "TON".TON[32].TON(pt := t#8s, et =>)
      S_Coil( "ST10_DeviceError".K.ReserveLine.UnloadingStop1timeout )
   END_RUNG
   // the same network as SCL:
   "TON".TON[32].TON(IN := "AlwaysTRUE" AND "ST10_Flow27_KReserveLoad&Unload_iDB".WaitPalletArrveNextPos_4.X AND NOT "iK-reserveTakeDetection2",
                     PT := t#8s);
   IF "TON".TON[32].Q THEN "ST10_DeviceError".K.ReserveLine.UnloadingStop1timeout := TRUE; END_IF;
END_REGION

REGION Network 85: unLoading Stop2 timeout
   RUNG wire#powerrail
      Contact( "AlwaysTRUE" )
      Contact( "ST10_Flow27_KReserveLoad&Unload_iDB".WaitPalletArrveNextPos_5.X )
      I_Contact( "iK-reserveTakeDetection3" )
      { S7_Templates := "time_type := Time" } "TON".TON[33].TON(pt := t#8s, et =>)
      S_Coil( "ST10_DeviceError".K.ReserveLine.UnloadingStop2timeout )
   END_RUNG
   // the same network as SCL:
   "TON".TON[33].TON(IN := "AlwaysTRUE" AND "ST10_Flow27_KReserveLoad&Unload_iDB".WaitPalletArrveNextPos_5.X AND NOT "iK-reserveTakeDetection3",
                     PT := t#8s);
   IF "TON".TON[33].Q THEN "ST10_DeviceError".K.ReserveLine.UnloadingStop2timeout := TRUE; END_IF;
END_REGION

REGION Network 86: unLoading Stop3 timeout
   RUNG wire#powerrail
      Contact( "AlwaysTRUE" )
      Contact( "ST10_Flow27_KReserveLoad&Unload_iDB".WaitPalletArrveNextPos_6.X )
      I_Contact( "iK-reserveTakeShaftDetection" )
      { S7_Templates := "time_type := Time" } "TON".TON[34].TON(pt := t#8s, et =>)
      S_Coil( "ST10_DeviceError".K.ReserveLine.UnloadingStop3timeout )
   END_RUNG
   // the same network as SCL:
   "TON".TON[34].TON(IN := "AlwaysTRUE" AND "ST10_Flow27_KReserveLoad&Unload_iDB".WaitPalletArrveNextPos_6.X AND NOT "iK-reserveTakeShaftDetection",
                     PT := t#8s);
   IF "TON".TON[34].Q THEN "ST10_DeviceError".K.ReserveLine.UnloadingStop3timeout := TRUE; END_IF;
END_REGION

REGION Network 87: Loading Lifting timeout
   RUNG wire#powerrail
      Contact( "AlwaysTRUE" )
      Contact( "ST10_Flow23_KReserveLifting_iDB".MotorCCWRun.X )
      I_Contact( "iK-reserveTakeDetection1" )
      { S7_Templates := "time_type := Time" } "TON".TON[35].TON(pt := t#8s, et =>)
      S_Coil( "ST10_DeviceError".K.ReserveLine.UnloadingLiftingtimeout )
   END_RUNG
   // the same network as SCL:
   "TON".TON[35].TON(IN := "AlwaysTRUE" AND "ST10_Flow23_KReserveLifting_iDB".MotorCCWRun.X AND NOT "iK-reserveTakeDetection1",
                     PT := t#8s);
   IF "TON".TON[35].Q THEN "ST10_DeviceError".K.ReserveLine.UnloadingLiftingtimeout := TRUE; END_IF;
END_REGION

REGION Network 88: Empty Stop1 timeout
   RUNG wire#powerrail
      Contact( "AlwaysTRUE" )
      Contact( "ST10_Flow27_KReserveLoad&Unload_iDB".WaitPalletArrveNextPos_10.X )
      I_Contact( "K-reservePalletEmptyCheck3" )
      { S7_Templates := "time_type := Time" } "TON".TON[36].TON(pt := t#8s, et =>)
      S_Coil( "ST10_DeviceError".K.ReserveLine.EmptyStop1timeout )
   END_RUNG
   // the same network as SCL:
   "TON".TON[36].TON(IN := "AlwaysTRUE" AND "ST10_Flow27_KReserveLoad&Unload_iDB".WaitPalletArrveNextPos_10.X AND NOT "K-reservePalletEmptyCheck3",
                     PT := t#8s);
   IF "TON".TON[36].Q THEN "ST10_DeviceError".K.ReserveLine.EmptyStop1timeout := TRUE; END_IF;
END_REGION

REGION Network 89: Empty Stop2 timeout
   RUNG wire#powerrail
      Contact( "AlwaysTRUE" )
      Contact( "ST10_Flow27_KReserveLoad&Unload_iDB".WaitPalletArrveNextPos_9.X )
      I_Contact( "K-reservePalletEmptyCheck2" )
      { S7_Templates := "time_type := Time" } "TON".TON[37].TON(pt := t#8s, et =>)
      S_Coil( "ST10_DeviceError".K.ReserveLine.EmptyStop2timeout )
   END_RUNG
   // the same network as SCL:
   "TON".TON[37].TON(IN := "AlwaysTRUE" AND "ST10_Flow27_KReserveLoad&Unload_iDB".WaitPalletArrveNextPos_9.X AND NOT "K-reservePalletEmptyCheck2",
                     PT := t#8s);
   IF "TON".TON[37].Q THEN "ST10_DeviceError".K.ReserveLine.EmptyStop2timeout := TRUE; END_IF;
END_REGION

REGION Network 90: Empty Stop3 timeout
   RUNG wire#powerrail
      Contact( "AlwaysTRUE" )
      Contact( "ST10_Flow27_KReserveLoad&Unload_iDB".WaitPalletArrveNextPos_8.X )
      I_Contact( "K-reservePalletEmptyCheck1" )
      { S7_Templates := "time_type := Time" } "TON".TON[38].TON(pt := t#8s, et =>)
      S_Coil( "ST10_DeviceError".K.ReserveLine.EmptyStop3timeout )
   END_RUNG
   // the same network as SCL:
   "TON".TON[38].TON(IN := "AlwaysTRUE" AND "ST10_Flow27_KReserveLoad&Unload_iDB".WaitPalletArrveNextPos_8.X AND NOT "K-reservePalletEmptyCheck1",
                     PT := t#8s);
   IF "TON".TON[38].Q THEN "ST10_DeviceError".K.ReserveLine.EmptyStop3timeout := TRUE; END_IF;
END_REGION

REGION Network 91: Empty Stop4 timeout
   RUNG wire#powerrail
      Contact( "AlwaysTRUE" )
      Contact( "ST10_Flow27_KReserveLoad&Unload_iDB".WaitPalletArrveNextPos_7.X )
      I_Contact( "iK-reserveTakeGateDetection" )
      { S7_Templates := "time_type := Time" } "TON".TON[39].TON(pt := t#8s, et =>)
      S_Coil( "ST10_DeviceError".K.ReserveLine.EmptyStop4timeout )
   END_RUNG
   // the same network as SCL:
   "TON".TON[39].TON(IN := "AlwaysTRUE" AND "ST10_Flow27_KReserveLoad&Unload_iDB".WaitPalletArrveNextPos_7.X AND NOT "iK-reserveTakeGateDetection",
                     PT := t#8s);
   IF "TON".TON[39].Q THEN "ST10_DeviceError".K.ReserveLine.EmptyStop4timeout := TRUE; END_IF;
END_REGION

REGION Network 93: ******************** L_Unloading ********************
END_REGION

REGION Network 94: L
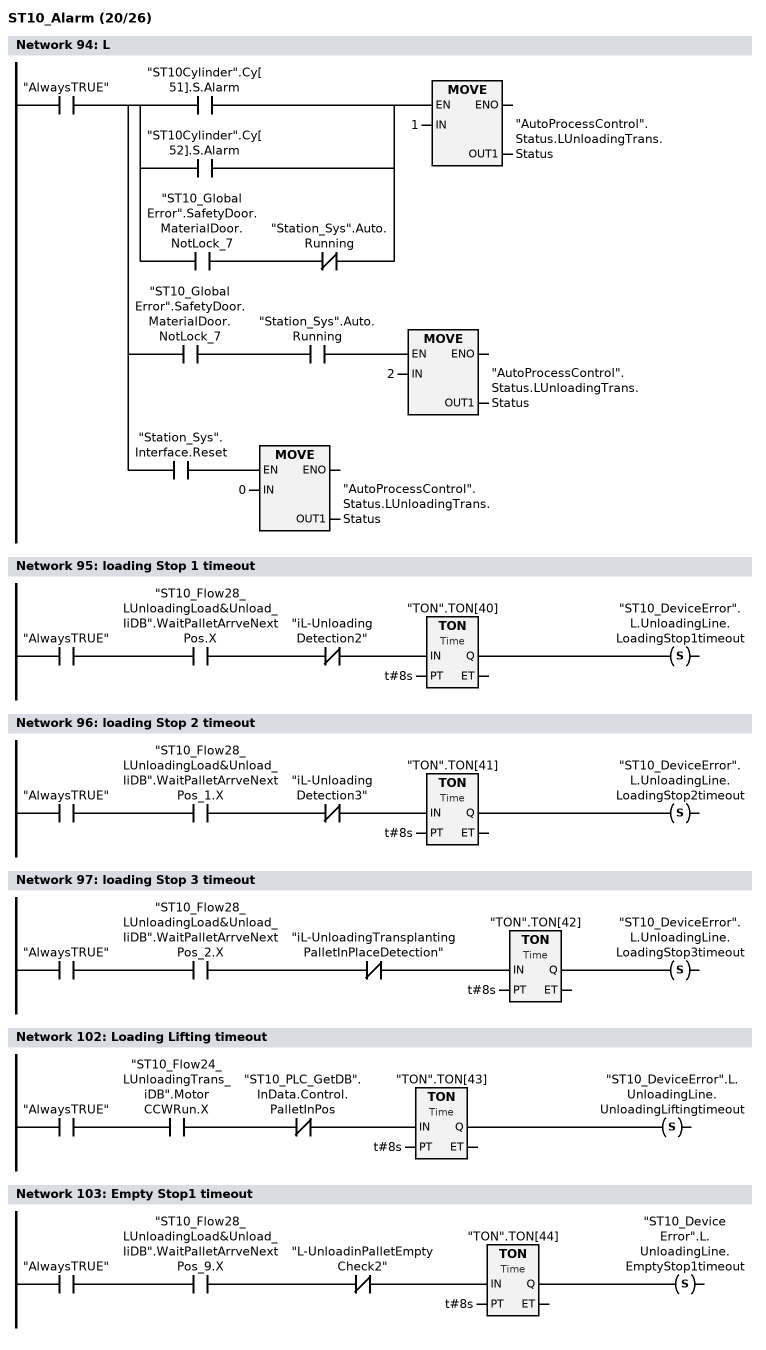
   RUNG wire#powerrail
      Contact( "AlwaysTRUE" )
      wire#w1
      Contact( "ST10Cylinder".Cy[51].S.Alarm )
      wire#w2
      Move(in := 1, out1 => "AutoProcessControl".Status.LUnloadingTrans.Status)
   END_RUNG
   RUNG wire#w1
      Contact( "ST10Cylinder".Cy[52].S.Alarm )
   END_RUNG wire#w2
   RUNG wire#w1
      Contact( "ST10_GlobalError".SafetyDoor.MaterialDoor.NotLock_7 )
      I_Contact( "Station_Sys".Auto.Running )
   END_RUNG wire#w2
   RUNG wire#w1
      Contact( "ST10_GlobalError".SafetyDoor.MaterialDoor.NotLock_7 )
      Contact( "Station_Sys".Auto.Running )
      Move(in := 2, out1 => "AutoProcessControl".Status.LUnloadingTrans.Status)
   END_RUNG
   RUNG wire#w1
      Contact( "Station_Sys".Interface.Reset )
      Move(in := 0, out1 => "AutoProcessControl".Status.LUnloadingTrans.Status)
   END_RUNG
   // the same network as SCL:
   IF "AlwaysTRUE" AND ("ST10Cylinder".Cy[51].S.Alarm OR "ST10Cylinder".Cy[52].S.Alarm OR ("ST10_GlobalError".SafetyDoor.MaterialDoor.NotLock_7 AND NOT "Station_Sys".Auto.Running)) THEN
       "AutoProcessControl".Status.LUnloadingTrans.Status := 1;
   END_IF;
   IF "AlwaysTRUE" AND "ST10_GlobalError".SafetyDoor.MaterialDoor.NotLock_7 AND "Station_Sys".Auto.Running THEN
       "AutoProcessControl".Status.LUnloadingTrans.Status := 2;
   END_IF;
   IF "AlwaysTRUE" AND "Station_Sys".Interface.Reset THEN
       "AutoProcessControl".Status.LUnloadingTrans.Status := 0;
   END_IF;
END_REGION

REGION Network 95: loading Stop 1 timeout
   RUNG wire#powerrail
      Contact( "AlwaysTRUE" )
      Contact( "ST10_Flow28_LUnloadingLoad&Unload_IiDB".WaitPalletArrveNextPos.X )
      I_Contact( "iL-UnloadingDetection2" )
      { S7_Templates := "time_type := Time" } "TON".TON[40].TON(pt := t#8s, et =>)
      S_Coil( "ST10_DeviceError".L.UnloadingLine.LoadingStop1timeout )
   END_RUNG
   // the same network as SCL:
   "TON".TON[40].TON(IN := "AlwaysTRUE" AND "ST10_Flow28_LUnloadingLoad&Unload_IiDB".WaitPalletArrveNextPos.X AND NOT "iL-UnloadingDetection2",
                     PT := t#8s);
   IF "TON".TON[40].Q THEN "ST10_DeviceError".L.UnloadingLine.LoadingStop1timeout := TRUE; END_IF;
END_REGION

REGION Network 96: loading Stop 2 timeout
   RUNG wire#powerrail
      Contact( "AlwaysTRUE" )
      Contact( "ST10_Flow28_LUnloadingLoad&Unload_IiDB".WaitPalletArrveNextPos_1.X )
      I_Contact( "iL-UnloadingDetection3" )
      { S7_Templates := "time_type := Time" } "TON".TON[41].TON(pt := t#8s, et =>)
      S_Coil( "ST10_DeviceError".L.UnloadingLine.LoadingStop2timeout )
   END_RUNG
   // the same network as SCL:
   "TON".TON[41].TON(IN := "AlwaysTRUE" AND "ST10_Flow28_LUnloadingLoad&Unload_IiDB".WaitPalletArrveNextPos_1.X AND NOT "iL-UnloadingDetection3",
                     PT := t#8s);
   IF "TON".TON[41].Q THEN "ST10_DeviceError".L.UnloadingLine.LoadingStop2timeout := TRUE; END_IF;
END_REGION

REGION Network 97: loading Stop 3 timeout
   RUNG wire#powerrail
      Contact( "AlwaysTRUE" )
      Contact( "ST10_Flow28_LUnloadingLoad&Unload_IiDB".WaitPalletArrveNextPos_2.X )
      I_Contact( "iL-UnloadingTransplantingPalletInPlaceDetection" )
      { S7_Templates := "time_type := Time" } "TON".TON[42].TON(pt := t#8s, et =>)
      S_Coil( "ST10_DeviceError".L.UnloadingLine.LoadingStop3timeout )
   END_RUNG
   // the same network as SCL:
   "TON".TON[42].TON(IN := "AlwaysTRUE" AND "ST10_Flow28_LUnloadingLoad&Unload_IiDB".WaitPalletArrveNextPos_2.X AND NOT "iL-UnloadingTransplantingPalletInPlaceDetection",
                     PT := t#8s);
   IF "TON".TON[42].Q THEN "ST10_DeviceError".L.UnloadingLine.LoadingStop3timeout := TRUE; END_IF;
END_REGION

REGION Network 98: loading Stop 4 timeout
END_REGION

REGION Network 99: unLoading Stop1 timeout
END_REGION

REGION Network 100: unLoading Stop2 timeout
END_REGION

REGION Network 101: unLoading Stop3 timeout
END_REGION

REGION Network 102: Loading Lifting timeout
   RUNG wire#powerrail
      Contact( "AlwaysTRUE" )
      Contact( "ST10_Flow24_LUnloadingTrans_iDB".MotorCCWRun.X )
      I_Contact( "ST10_PLC_GetDB".InData.Control.PalletInPos )
      { S7_Templates := "time_type := Time" } "TON".TON[43].TON(pt := t#8s, et =>)
      S_Coil( "ST10_DeviceError".L.UnloadingLine.UnloadingLiftingtimeout )
   END_RUNG
   // the same network as SCL:
   "TON".TON[43].TON(IN := "AlwaysTRUE" AND "ST10_Flow24_LUnloadingTrans_iDB".MotorCCWRun.X AND NOT "ST10_PLC_GetDB".InData.Control.PalletInPos,
                     PT := t#8s);
   IF "TON".TON[43].Q THEN "ST10_DeviceError".L.UnloadingLine.UnloadingLiftingtimeout := TRUE; END_IF;
END_REGION

REGION Network 103: Empty Stop1 timeout
   RUNG wire#powerrail
      Contact( "AlwaysTRUE" )
      Contact( "ST10_Flow28_LUnloadingLoad&Unload_IiDB".WaitPalletArrveNextPos_9.X )
      I_Contact( "L-UnloadinPalletEmptyCheck2" )
      { S7_Templates := "time_type := Time" } "TON".TON[44].TON(pt := t#8s, et =>)
      S_Coil( "ST10_DeviceError".L.UnloadingLine.EmptyStop1timeout )
   END_RUNG
   // the same network as SCL:
   "TON".TON[44].TON(IN := "AlwaysTRUE" AND "ST10_Flow28_LUnloadingLoad&Unload_IiDB".WaitPalletArrveNextPos_9.X AND NOT "L-UnloadinPalletEmptyCheck2",
                     PT := t#8s);
   IF "TON".TON[44].Q THEN "ST10_DeviceError".L.UnloadingLine.EmptyStop1timeout := TRUE; END_IF;
END_REGION

REGION Network 104: Empty Stop2 timeout
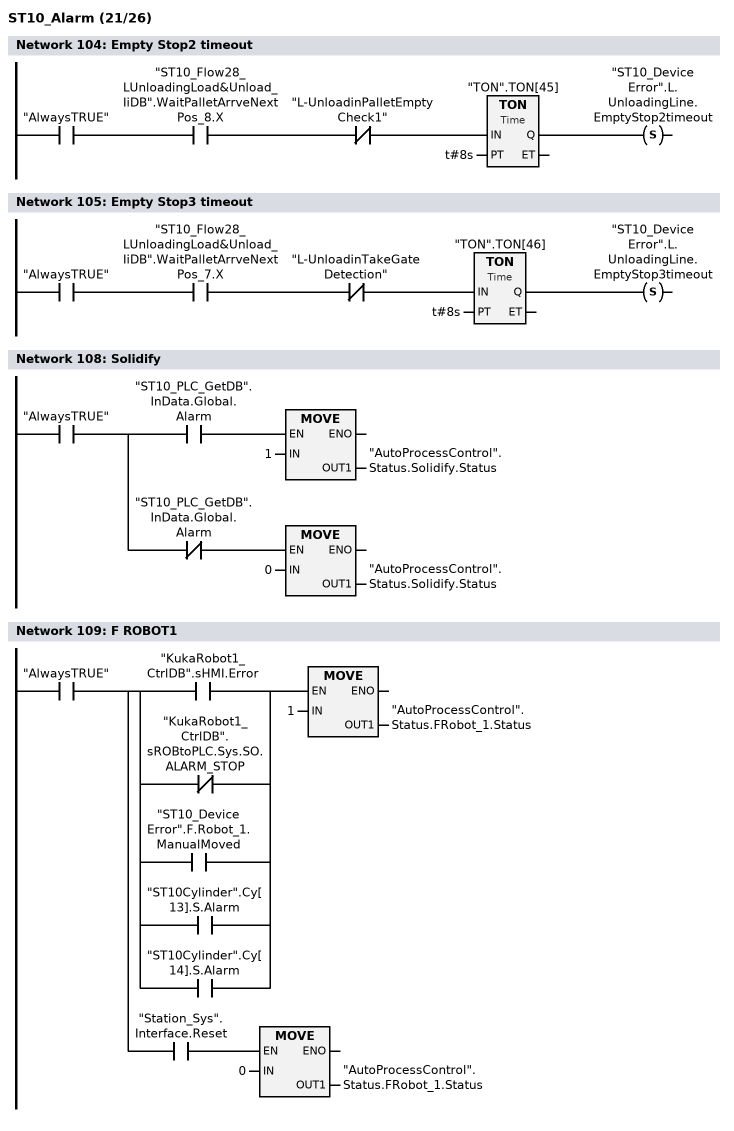
   RUNG wire#powerrail
      Contact( "AlwaysTRUE" )
      Contact( "ST10_Flow28_LUnloadingLoad&Unload_IiDB".WaitPalletArrveNextPos_8.X )
      I_Contact( "L-UnloadinPalletEmptyCheck1" )
      { S7_Templates := "time_type := Time" } "TON".TON[45].TON(pt := t#8s, et =>)
      S_Coil( "ST10_DeviceError".L.UnloadingLine.EmptyStop2timeout )
   END_RUNG
   // the same network as SCL:
   "TON".TON[45].TON(IN := "AlwaysTRUE" AND "ST10_Flow28_LUnloadingLoad&Unload_IiDB".WaitPalletArrveNextPos_8.X AND NOT "L-UnloadinPalletEmptyCheck1",
                     PT := t#8s);
   IF "TON".TON[45].Q THEN "ST10_DeviceError".L.UnloadingLine.EmptyStop2timeout := TRUE; END_IF;
END_REGION

REGION Network 105: Empty Stop3 timeout
   RUNG wire#powerrail
      Contact( "AlwaysTRUE" )
      Contact( "ST10_Flow28_LUnloadingLoad&Unload_IiDB".WaitPalletArrveNextPos_7.X )
      I_Contact( "L-UnloadinTakeGateDetection" )
      { S7_Templates := "time_type := Time" } "TON".TON[46].TON(pt := t#8s, et =>)
      S_Coil( "ST10_DeviceError".L.UnloadingLine.EmptyStop3timeout )
   END_RUNG
   // the same network as SCL:
   "TON".TON[46].TON(IN := "AlwaysTRUE" AND "ST10_Flow28_LUnloadingLoad&Unload_IiDB".WaitPalletArrveNextPos_7.X AND NOT "L-UnloadinTakeGateDetection",
                     PT := t#8s);
   IF "TON".TON[46].Q THEN "ST10_DeviceError".L.UnloadingLine.EmptyStop3timeout := TRUE; END_IF;
END_REGION

REGION Network 106: Empty Stop4 timeout
END_REGION

REGION Network 108: Solidify
   RUNG wire#powerrail
      Contact( "AlwaysTRUE" )
      wire#w1
      Contact( "ST10_PLC_GetDB".InData.Global.Alarm )
      Move(in := 1, out1 => "AutoProcessControl".Status.Solidify.Status)
   END_RUNG
   RUNG wire#w1
      I_Contact( "ST10_PLC_GetDB".InData.Global.Alarm )
      Move(in := 0, out1 => "AutoProcessControl".Status.Solidify.Status)
   END_RUNG
   // the same network as SCL:
   IF "AlwaysTRUE" AND "ST10_PLC_GetDB".InData.Global.Alarm THEN
       "AutoProcessControl".Status.Solidify.Status := 1;
   END_IF;
   IF "AlwaysTRUE" AND NOT "ST10_PLC_GetDB".InData.Global.Alarm THEN
       "AutoProcessControl".Status.Solidify.Status := 0;
   END_IF;
END_REGION

REGION Network 109: F ROBOT1
   RUNG wire#powerrail
      Contact( "AlwaysTRUE" )
      wire#w1
      Contact( "KukaRobot1_CtrlDB".sHMI.Error )
      wire#w2
      Move(in := 1, out1 => "AutoProcessControl".Status.FRobot_1.Status)
   END_RUNG
   RUNG wire#w1
      I_Contact( "KukaRobot1_CtrlDB".sROBtoPLC.Sys.SO.ALARM_STOP )
   END_RUNG wire#w2
   RUNG wire#w1
      Contact( "ST10_DeviceError".F.Robot_1.ManualMoved )
   END_RUNG wire#w2
   RUNG wire#w1
      Contact( "ST10Cylinder".Cy[13].S.Alarm )
   END_RUNG wire#w2
   RUNG wire#w1
      Contact( "ST10Cylinder".Cy[14].S.Alarm )
   END_RUNG wire#w2
   RUNG wire#w1
      Contact( "Station_Sys".Interface.Reset )
      Move(in := 0, out1 => "AutoProcessControl".Status.FRobot_1.Status)
   END_RUNG
   // the same network as SCL:
   IF "AlwaysTRUE" AND ("KukaRobot1_CtrlDB".sHMI.Error OR NOT "KukaRobot1_CtrlDB".sROBtoPLC.Sys.SO.ALARM_STOP OR "ST10_DeviceError".F.Robot_1.ManualMoved OR "ST10Cylinder".Cy[13].S.Alarm OR "ST10Cylinder".Cy[14].S.Alarm) THEN
       "AutoProcessControl".Status.FRobot_1.Status := 1;
   END_IF;
   IF "AlwaysTRUE" AND "Station_Sys".Interface.Reset THEN
       "AutoProcessControl".Status.FRobot_1.Status := 0;
   END_IF;
END_REGION

REGION Network 110: F ROBOT2
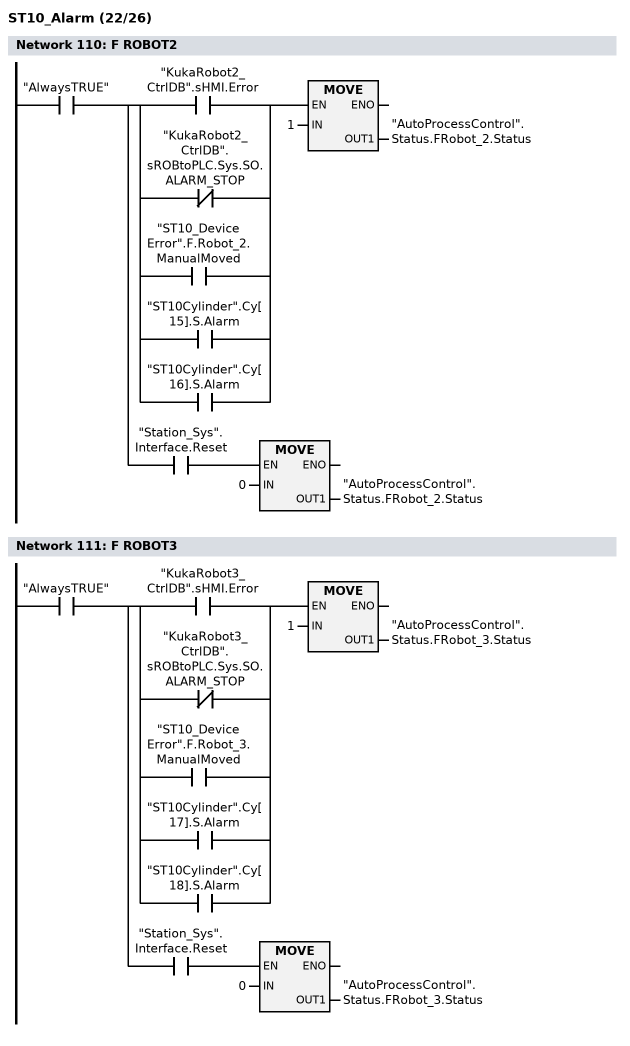
   RUNG wire#powerrail
      Contact( "AlwaysTRUE" )
      wire#w1
      Contact( "KukaRobot2_CtrlDB".sHMI.Error )
      wire#w2
      Move(in := 1, out1 => "AutoProcessControl".Status.FRobot_2.Status)
   END_RUNG
   RUNG wire#w1
      I_Contact( "KukaRobot2_CtrlDB".sROBtoPLC.Sys.SO.ALARM_STOP )
   END_RUNG wire#w2
   RUNG wire#w1
      Contact( "ST10_DeviceError".F.Robot_2.ManualMoved )
   END_RUNG wire#w2
   RUNG wire#w1
      Contact( "ST10Cylinder".Cy[15].S.Alarm )
   END_RUNG wire#w2
   RUNG wire#w1
      Contact( "ST10Cylinder".Cy[16].S.Alarm )
   END_RUNG wire#w2
   RUNG wire#w1
      Contact( "Station_Sys".Interface.Reset )
      Move(in := 0, out1 => "AutoProcessControl".Status.FRobot_2.Status)
   END_RUNG
   // the same network as SCL:
   IF "AlwaysTRUE" AND ("KukaRobot2_CtrlDB".sHMI.Error OR NOT "KukaRobot2_CtrlDB".sROBtoPLC.Sys.SO.ALARM_STOP OR "ST10_DeviceError".F.Robot_2.ManualMoved OR "ST10Cylinder".Cy[15].S.Alarm OR "ST10Cylinder".Cy[16].S.Alarm) THEN
       "AutoProcessControl".Status.FRobot_2.Status := 1;
   END_IF;
   IF "AlwaysTRUE" AND "Station_Sys".Interface.Reset THEN
       "AutoProcessControl".Status.FRobot_2.Status := 0;
   END_IF;
END_REGION

REGION Network 111: F ROBOT3
   RUNG wire#powerrail
      Contact( "AlwaysTRUE" )
      wire#w1
      Contact( "KukaRobot3_CtrlDB".sHMI.Error )
      wire#w2
      Move(in := 1, out1 => "AutoProcessControl".Status.FRobot_3.Status)
   END_RUNG
   RUNG wire#w1
      I_Contact( "KukaRobot3_CtrlDB".sROBtoPLC.Sys.SO.ALARM_STOP )
   END_RUNG wire#w2
   RUNG wire#w1
      Contact( "ST10_DeviceError".F.Robot_3.ManualMoved )
   END_RUNG wire#w2
   RUNG wire#w1
      Contact( "ST10Cylinder".Cy[17].S.Alarm )
   END_RUNG wire#w2
   RUNG wire#w1
      Contact( "ST10Cylinder".Cy[18].S.Alarm )
   END_RUNG wire#w2
   RUNG wire#w1
      Contact( "Station_Sys".Interface.Reset )
      Move(in := 0, out1 => "AutoProcessControl".Status.FRobot_3.Status)
   END_RUNG
   // the same network as SCL:
   IF "AlwaysTRUE" AND ("KukaRobot3_CtrlDB".sHMI.Error OR NOT "KukaRobot3_CtrlDB".sROBtoPLC.Sys.SO.ALARM_STOP OR "ST10_DeviceError".F.Robot_3.ManualMoved OR "ST10Cylinder".Cy[17].S.Alarm OR "ST10Cylinder".Cy[18].S.Alarm) THEN
       "AutoProcessControl".Status.FRobot_3.Status := 1;
   END_IF;
   IF "AlwaysTRUE" AND "Station_Sys".Interface.Reset THEN
       "AutoProcessControl".Status.FRobot_3.Status := 0;
   END_IF;
END_REGION

REGION Network 112: ******************** E NG ********************
END_REGION

REGION Network 113: E NG_1
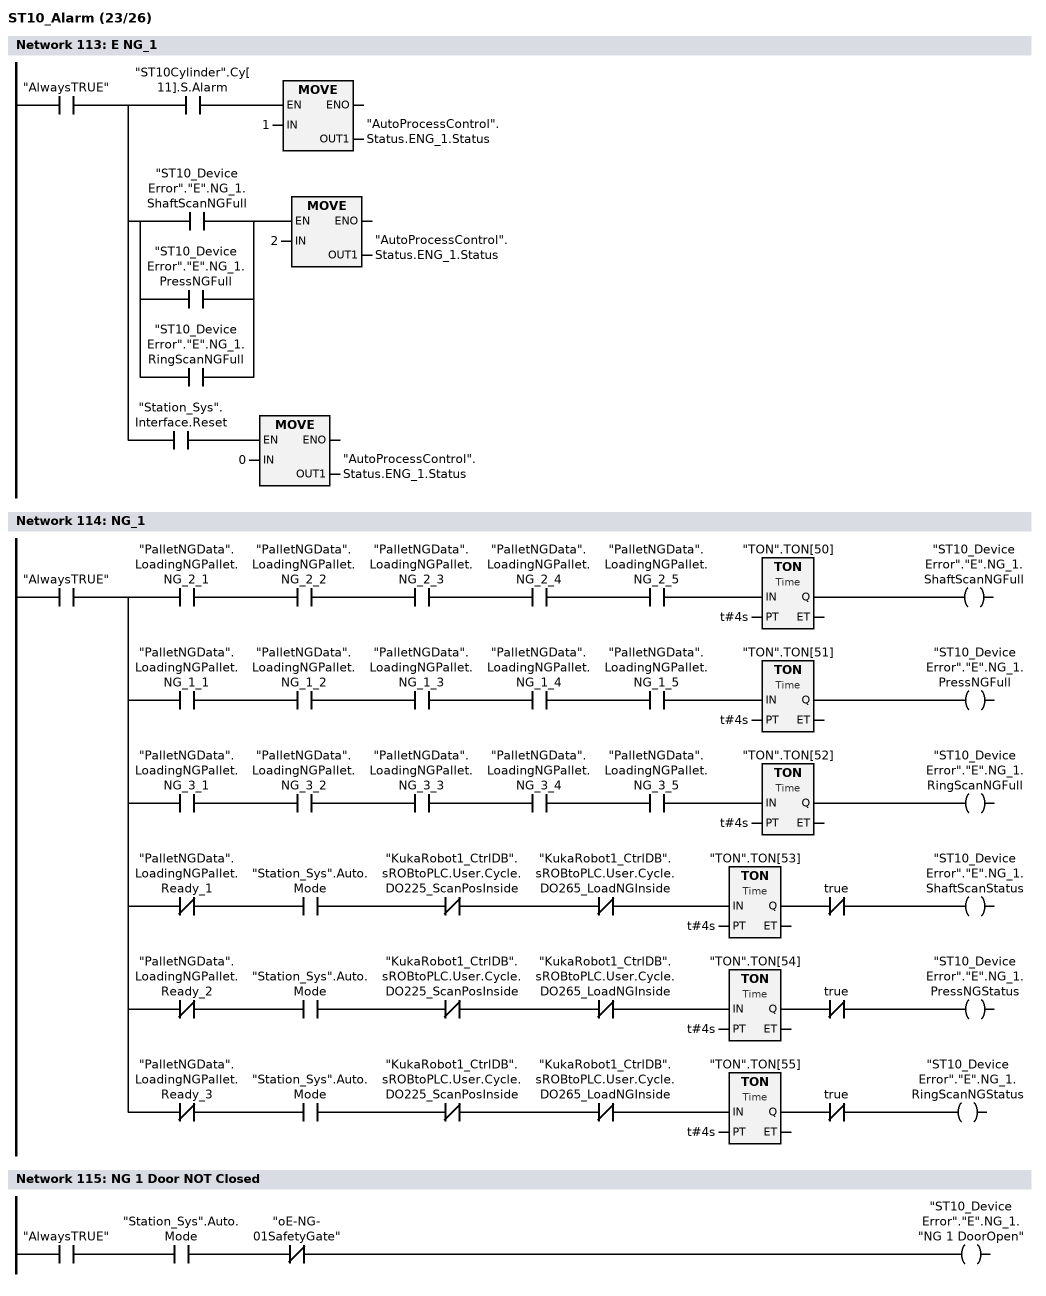
   RUNG wire#powerrail
      Contact( "AlwaysTRUE" )
      wire#w1
      Contact( "ST10Cylinder".Cy[11].S.Alarm )
      Move(in := 1, out1 => "AutoProcessControl".Status.ENG_1.Status)
   END_RUNG
   RUNG wire#w1
      Contact( "ST10_DeviceError"."E".NG_1.ShaftScanNGFull )
      wire#w2
      Move(in := 2, out1 => "AutoProcessControl".Status.ENG_1.Status)
   END_RUNG
   RUNG wire#w1
      Contact( "ST10_DeviceError"."E".NG_1.PressNGFull )
   END_RUNG wire#w2
   RUNG wire#w1
      Contact( "ST10_DeviceError"."E".NG_1.RingScanNGFull )
   END_RUNG wire#w2
   RUNG wire#w1
      Contact( "Station_Sys".Interface.Reset )
      Move(in := 0, out1 => "AutoProcessControl".Status.ENG_1.Status)
   END_RUNG
   // the same network as SCL:
   IF "AlwaysTRUE" AND "ST10Cylinder".Cy[11].S.Alarm THEN
       "AutoProcessControl".Status.ENG_1.Status := 1;
   END_IF;
   IF "AlwaysTRUE" AND ("ST10_DeviceError"."E".NG_1.ShaftScanNGFull OR "ST10_DeviceError"."E".NG_1.PressNGFull OR "ST10_DeviceError"."E".NG_1.RingScanNGFull) THEN
       "AutoProcessControl".Status.ENG_1.Status := 2;
   END_IF;
   IF "AlwaysTRUE" AND "Station_Sys".Interface.Reset THEN
       "AutoProcessControl".Status.ENG_1.Status := 0;
   END_IF;
END_REGION

REGION Network 114: NG_1
   RUNG wire#powerrail
      Contact( "AlwaysTRUE" )
      wire#w1
      Contact( "PalletNGData".LoadingNGPallet.NG_2_1 )
      Contact( "PalletNGData".LoadingNGPallet.NG_2_2 )
      Contact( "PalletNGData".LoadingNGPallet.NG_2_3 )
      Contact( "PalletNGData".LoadingNGPallet.NG_2_4 )
      Contact( "PalletNGData".LoadingNGPallet.NG_2_5 )
      { S7_Templates := "time_type := Time" } "TON".TON[50].TON(pt := t#4s, et =>)
      Coil( "ST10_DeviceError"."E".NG_1.ShaftScanNGFull )
   END_RUNG
   RUNG wire#w1
      Contact( "PalletNGData".LoadingNGPallet.NG_1_1 )
      Contact( "PalletNGData".LoadingNGPallet.NG_1_2 )
      Contact( "PalletNGData".LoadingNGPallet.NG_1_3 )
      Contact( "PalletNGData".LoadingNGPallet.NG_1_4 )
      Contact( "PalletNGData".LoadingNGPallet.NG_1_5 )
      { S7_Templates := "time_type := Time" } "TON".TON[51].TON(pt := t#4s, et =>)
      Coil( "ST10_DeviceError"."E".NG_1.PressNGFull )
   END_RUNG
   RUNG wire#w1
      Contact( "PalletNGData".LoadingNGPallet.NG_3_1 )
      Contact( "PalletNGData".LoadingNGPallet.NG_3_2 )
      Contact( "PalletNGData".LoadingNGPallet.NG_3_3 )
      Contact( "PalletNGData".LoadingNGPallet.NG_3_4 )
      Contact( "PalletNGData".LoadingNGPallet.NG_3_5 )
      { S7_Templates := "time_type := Time" } "TON".TON[52].TON(pt := t#4s, et =>)
      Coil( "ST10_DeviceError"."E".NG_1.RingScanNGFull )
   END_RUNG
   RUNG wire#w1
      I_Contact( "PalletNGData".LoadingNGPallet.Ready_1 )
      Contact( "Station_Sys".Auto.Mode )
      I_Contact( "KukaRobot1_CtrlDB".sROBtoPLC.User.Cycle.DO225_ScanPosInside )
      I_Contact( "KukaRobot1_CtrlDB".sROBtoPLC.User.Cycle.DO265_LoadNGInside )
      { S7_Templates := "time_type := Time" } "TON".TON[53].TON(pt := t#4s, et =>)
      I_Contact( true )
      Coil( "ST10_DeviceError"."E".NG_1.ShaftScanStatus )
   END_RUNG
   RUNG wire#w1
      I_Contact( "PalletNGData".LoadingNGPallet.Ready_2 )
      Contact( "Station_Sys".Auto.Mode )
      I_Contact( "KukaRobot1_CtrlDB".sROBtoPLC.User.Cycle.DO225_ScanPosInside )
      I_Contact( "KukaRobot1_CtrlDB".sROBtoPLC.User.Cycle.DO265_LoadNGInside )
      { S7_Templates := "time_type := Time" } "TON".TON[54].TON(pt := t#4s, et =>)
      I_Contact( true )
      Coil( "ST10_DeviceError"."E".NG_1.PressNGStatus )
   END_RUNG
   RUNG wire#w1
      I_Contact( "PalletNGData".LoadingNGPallet.Ready_3 )
      Contact( "Station_Sys".Auto.Mode )
      I_Contact( "KukaRobot1_CtrlDB".sROBtoPLC.User.Cycle.DO225_ScanPosInside )
      I_Contact( "KukaRobot1_CtrlDB".sROBtoPLC.User.Cycle.DO265_LoadNGInside )
      { S7_Templates := "time_type := Time" } "TON".TON[55].TON(pt := t#4s, et =>)
      I_Contact( true )
      Coil( "ST10_DeviceError"."E".NG_1.RingScanNGStatus )
   END_RUNG
   // the same network as SCL:
   "TON".TON[50].TON(IN := "AlwaysTRUE" AND "PalletNGData".LoadingNGPallet.NG_2_1 AND "PalletNGData".LoadingNGPallet.NG_2_2 AND "PalletNGData".LoadingNGPallet.NG_2_3 AND "PalletNGData".LoadingNGPallet.NG_2_4 AND "PalletNGData".LoadingNGPallet.NG_2_5,
                     PT := t#4s);
   "ST10_DeviceError"."E".NG_1.ShaftScanNGFull := "TON".TON[50].Q;
   "TON".TON[51].TON(IN := "AlwaysTRUE" AND "PalletNGData".LoadingNGPallet.NG_1_1 AND "PalletNGData".LoadingNGPallet.NG_1_2 AND "PalletNGData".LoadingNGPallet.NG_1_3 AND "PalletNGData".LoadingNGPallet.NG_1_4 AND "PalletNGData".LoadingNGPallet.NG_1_5,
                     PT := t#4s);
   "ST10_DeviceError"."E".NG_1.PressNGFull := "TON".TON[51].Q;
   "TON".TON[52].TON(IN := "AlwaysTRUE" AND "PalletNGData".LoadingNGPallet.NG_3_1 AND "PalletNGData".LoadingNGPallet.NG_3_2 AND "PalletNGData".LoadingNGPallet.NG_3_3 AND "PalletNGData".LoadingNGPallet.NG_3_4 AND "PalletNGData".LoadingNGPallet.NG_3_5,
                     PT := t#4s);
   "ST10_DeviceError"."E".NG_1.RingScanNGFull := "TON".TON[52].Q;
   "TON".TON[53].TON(IN := "AlwaysTRUE" AND NOT "PalletNGData".LoadingNGPallet.Ready_1 AND "Station_Sys".Auto.Mode AND NOT "KukaRobot1_CtrlDB".sROBtoPLC.User.Cycle.DO225_ScanPosInside AND NOT "KukaRobot1_CtrlDB".sROBtoPLC.User.Cycle.DO265_LoadNGInside,
                     PT := t#4s);
   "ST10_DeviceError"."E".NG_1.ShaftScanStatus := "TON".TON[53].Q AND NOT true;
   "TON".TON[54].TON(IN := "AlwaysTRUE" AND NOT "PalletNGData".LoadingNGPallet.Ready_2 AND "Station_Sys".Auto.Mode AND NOT "KukaRobot1_CtrlDB".sROBtoPLC.User.Cycle.DO225_ScanPosInside AND NOT "KukaRobot1_CtrlDB".sROBtoPLC.User.Cycle.DO265_LoadNGInside,
                     PT := t#4s);
   "ST10_DeviceError"."E".NG_1.PressNGStatus := "TON".TON[54].Q AND NOT true;
   "TON".TON[55].TON(IN := "AlwaysTRUE" AND NOT "PalletNGData".LoadingNGPallet.Ready_3 AND "Station_Sys".Auto.Mode AND NOT "KukaRobot1_CtrlDB".sROBtoPLC.User.Cycle.DO225_ScanPosInside AND NOT "KukaRobot1_CtrlDB".sROBtoPLC.User.Cycle.DO265_LoadNGInside,
                     PT := t#4s);
   "ST10_DeviceError"."E".NG_1.RingScanNGStatus := "TON".TON[55].Q AND NOT true;
END_REGION

